Yaskawa INFORM job: BLACKRUN.JBI

/JOB
//NAME BLACKRUN
//POS
///NPOS 4041,0,0,0,0,0
///TOOL 0
///POSTYPE PULSE
///PULSE
C00000=-2822,58859,-1118,-1041,-34109,-89
C00001=-2591,62265,5411,-1016,-36162,-226
C00002=-2591,62265,4011,-1016,-36162,-226
C00003=-2454,62257,4002,-1034,-36158,-281
C00004=-2454,62257,5402,-1034,-36158,-281
C00005=-2634,62224,5347,-1011,-36136,-208
C00006=-2634,62224,3947,-1011,-36136,-208
C00007=-2403,62210,3931,-1041,-36129,-301
C00008=-2403,62210,5331,-1041,-36129,-301
C00009=-2660,62181,5282,-1008,-36110,-197
C00010=-2660,62181,3882,-1008,-36110,-197
C00011=-2607,62178,3878,-1015,-36108,-219
C00012=-2607,62178,5278,-1015,-36108,-219
C00013=-2442,62168,5267,-1037,-36104,-285
C00014=-2442,62168,3867,-1037,-36104,-285
C00015=-2393,62165,3864,-1043,-36102,-305
C00016=-2393,62165,5264,-1043,-36102,-305
C00017=-4693,62262,5357,-741,-36142,620
C00018=-4693,62262,3957,-741,-36142,620
C00019=-4619,62257,3952,-751,-36140,591
C00020=-4619,62257,5352,-751,-36140,591
C00021=-4342,62240,5333,-787,-36132,479
C00022=-4342,62240,3933,-787,-36132,479
C00023=-3994,62219,3908,-833,-36122,340
C00024=-3994,62219,5308,-833,-36122,340
C00025=-2682,62138,5217,-1006,-36083,-188
C00026=-2682,62138,3817,-1006,-36083,-188
C00027=-2632,62135,3813,-1012,-36082,-208
C00028=-2632,62135,5213,-1012,-36082,-208
C00029=-2432,62123,5199,-1039,-36076,-288
C00030=-2432,62123,3799,-1039,-36076,-288
C00031=-2387,62120,3796,-1045,-36075,-307
C00032=-2387,62120,5196,-1045,-36075,-307
C00033=-4830,62226,5300,-724,-36119,676
C00034=-4830,62226,3900,-724,-36119,676
C00035=-4543,62208,3880,-762,-36110,560
C00036=-4543,62208,5280,-762,-36110,560
C00037=-4469,62203,5275,-771,-36108,531
C00038=-4469,62203,3875,-771,-36108,531
C00039=-4244,62190,3859,-801,-36102,441
C00040=-4244,62190,5259,-801,-36102,441
C00041=-4090,62180,5248,-821,-36097,379
C00042=-4090,62180,3848,-821,-36097,379
C00043=-3855,62166,3832,-852,-36090,284
C00044=-3855,62166,5232,-852,-36090,284
C00045=-2696,62095,5151,-1005,-36057,-182
C00046=-2696,62095,3751,-1005,-36057,-182
C00047=-2654,62092,3748,-1010,-36056,-198
C00048=-2654,62092,5148,-1010,-36056,-198
C00049=-2423,62078,5132,-1041,-36049,-292
C00050=-2423,62078,3732,-1041,-36049,-292
C00051=-2381,62075,3729,-1046,-36048,-309
C00052=-2381,62075,5129,-1046,-36048,-309
C00053=-4912,62186,5238,-714,-36094,710
C00054=-4912,62186,3838,-714,-36094,710
C00055=-4782,62178,3829,-731,-36090,657
C00056=-4782,62178,5229,-731,-36090,657
C00057=-4596,62167,5216,-755,-36085,583
C00058=-4596,62167,3816,-755,-36085,583
C00059=-4445,62157,3806,-775,-36081,522
C00060=-4445,62157,5206,-775,-36081,522
C00061=-3929,62126,5170,-843,-36066,315
C00062=-3929,62126,3770,-843,-36066,315
C00063=-3778,62117,3759,-863,-36061,254
C00064=-3778,62117,5159,-863,-36061,254
C00065=-2708,62051,5084,-1004,-36030,-176
C00066=-2708,62051,3684,-1004,-36030,-176
C00067=-2673,62049,3682,-1008,-36029,-191
C00068=-2673,62049,5082,-1008,-36029,-191
C00069=-2413,62033,5064,-1043,-36022,-295
C00070=-2413,62033,3664,-1043,-36022,-295
C00071=-2371,62031,3661,-1048,-36020,-312
C00072=-2371,62031,5061,-1048,-36020,-312
C00073=-4976,62146,5176,-706,-36069,736
C00074=-4976,62146,3776,-706,-36069,736
C00075=-4864,62139,3768,-721,-36066,691
C00076=-4864,62139,5168,-721,-36066,691
C00077=-4713,62129,5157,-740,-36062,630
C00078=-4713,62129,3757,-740,-36062,630
C00079=-4576,62121,3748,-758,-36058,575
C00080=-4576,62121,5148,-758,-36058,575
C00081=-4488,62116,5142,-770,-36055,540
C00082=-4488,62116,3742,-770,-36055,540
C00083=-4415,62111,3737,-780,-36053,510
C00084=-4415,62111,5137,-780,-36053,510
C00085=-3821,62075,5095,-858,-36036,272
C00086=-3821,62075,3695,-858,-36036,272
C00087=-3713,62068,3688,-872,-36032,228
C00088=-3713,62068,5088,-872,-36032,228
C00089=-2726,62008,5019,-1002,-36004,-168
C00090=-2726,62008,3619,-1002,-36004,-168
C00091=-2688,62006,3616,-1007,-36003,-184
C00092=-2688,62006,5016,-1007,-36003,-184
C00093=-2407,61988,4996,-1044,-35994,-297
C00094=-2407,61988,3596,-1044,-35994,-297
C00095=-2361,61986,3593,-1050,-35993,-315
C00096=-2361,61986,4993,-1050,-35993,-315
C00097=-5012,62103,5111,-702,-36043,751
C00098=-5012,62103,3711,-702,-36043,751
C00099=-4928,62098,3705,-713,-36041,717
C00100=-4928,62098,5105,-713,-36041,717
C00101=-3752,62026,5023,-868,-36007,244
C00102=-3752,62026,3623,-868,-36007,244
C00103=-3661,62021,3617,-880,-36004,208
C00104=-3661,62021,5017,-880,-36004,208
C00105=-2738,61964,4952,-1001,-35977,-163
C00106=-2738,61964,3552,-1001,-35977,-163
C00107=-2699,61962,3550,-1006,-35976,-179
C00108=-2699,61962,4950,-1006,-35976,-179
C00109=-2401,61944,4929,-1046,-35967,-299
C00110=-2401,61944,3529,-1046,-35967,-299
C00111=-2355,61941,3526,-1052,-35966,-317
C00112=-2355,61941,4926,-1052,-35966,-317
C00113=-5056,62061,5047,-697,-36018,769
C00114=-5056,62061,3647,-697,-36018,769
C00115=-4985,62057,3642,-706,-36016,741
C00116=-4985,62057,5042,-706,-36016,741
C00117=-3697,61979,4952,-876,-35978,223
C00118=-3697,61979,3552,-876,-35978,223
C00119=-3630,61975,3548,-884,-35976,196
C00120=-3630,61975,4948,-884,-35976,196
C00121=-2745,61921,4886,-1001,-35950,-160
C00122=-2745,61921,3486,-1001,-35950,-160
C00123=-2714,61919,3484,-1005,-35949,-172
C00124=-2714,61919,4884,-1005,-35949,-172
C00125=-2398,61899,4862,-1047,-35940,-299
C00126=-2398,61899,3462,-1047,-35940,-299
C00127=-2352,61897,3458,-1053,-35939,-318
C00128=-2352,61897,4858,-1053,-35939,-318
C00129=-5099,62020,4983,-692,-35992,787
C00130=-5099,62020,3583,-692,-35992,787
C00131=-5025,62015,3578,-701,-35990,757
C00132=-5025,62015,4978,-701,-35990,757
C00133=-3656,61932,4882,-882,-35950,207
C00134=-3656,61932,3482,-882,-35950,207
C00135=-3603,61929,3479,-889,-35948,186
C00136=-3603,61929,4879,-889,-35948,186
C00137=-2750,61877,4819,-1001,-35923,-157
C00138=-2750,61877,3419,-1001,-35923,-157
C00139=-2722,61875,3417,-1005,-35922,-169
C00140=-2722,61875,4817,-1005,-35922,-169
C00141=-2392,61855,4794,-1048,-35913,-301
C00142=-2392,61855,3394,-1048,-35913,-301
C00143=-2343,61852,3391,-1055,-35911,-321
C00144=-2343,61852,4791,-1055,-35911,-321
C00145=126,61702,4618,-1380,-35839,-1313
C00146=126,61702,3218,-1380,-35839,-1313
C00147=150,61700,3217,-1383,-35838,-1323
C00148=150,61700,4617,-1383,-35838,-1323
C00149=-5135,61977,4919,-688,-35966,802
C00150=-5135,61977,3519,-688,-35966,802
C00151=-5065,61973,3514,-697,-35964,773
C00152=-5065,61973,4914,-697,-35964,773
C00153=-3632,61886,4814,-886,-35922,198
C00154=-3632,61886,3414,-886,-35922,198
C00155=-3565,61882,3409,-894,-35920,171
C00156=-3565,61882,4809,-894,-35920,171
C00157=-2758,61833,4753,-1001,-35896,-154
C00158=-2758,61833,3353,-1001,-35896,-154
C00159=-2726,61831,3350,-1005,-35896,-166
C00160=-2726,61831,4750,-1005,-35896,-166
C00161=-2389,61810,4727,-1049,-35886,-302
C00162=-2389,61810,3327,-1049,-35886,-302
C00163=-2350,61808,3324,-1055,-35884,-317
C00164=-2350,61808,4724,-1055,-35884,-317
C00165=-935,61722,4625,-1241,-35843,-886
C00166=-935,61722,3225,-1241,-35843,-886
C00167=-890,61719,3222,-1247,-35842,-904
C00168=-890,61719,4622,-1247,-35842,-904
C00169=128,61657,4551,-1381,-35812,-1313
C00170=128,61657,3151,-1381,-35812,-1313
C00171=171,61655,3148,-1387,-35811,-1330
C00172=171,61655,4548,-1387,-35811,-1330
C00173=-5164,61935,4854,-684,-35940,814
C00174=-5164,61935,3454,-684,-35940,814
C00175=-5104,61931,3449,-692,-35938,790
C00176=-5104,61931,4849,-692,-35938,790
C00177=-3601,61840,4744,-890,-35894,186
C00178=-3601,61840,3344,-890,-35894,186
C00179=-3528,61835,3339,-900,-35892,156
C00180=-3528,61835,4739,-900,-35892,156
C00181=-2766,61789,4686,-1001,-35870,-150
C00182=-2766,61789,3286,-1001,-35870,-150
C00183=-2730,61787,3284,-1005,-35869,-164
C00184=-2730,61787,4684,-1005,-35869,-164
C00185=-936,61678,4558,-1242,-35816,-885
C00186=-936,61678,3158,-1242,-35816,-885
C00187=-891,61675,3155,-1248,-35815,-903
C00188=-891,61675,4555,-1248,-35815,-903
C00189=-747,61666,4545,-1267,-35810,-961
C00190=-747,61666,3145,-1267,-35810,-961
C00191=-704,61664,3142,-1272,-35809,-978
C00192=-704,61664,4542,-1272,-35809,-978
C00193=142,61613,4483,-1384,-35784,-1318
C00194=142,61613,3083,-1384,-35784,-1318
C00195=180,61610,3080,-1389,-35783,-1333
C00196=180,61610,4480,-1389,-35783,-1333
C00197=-5196,61892,4789,-681,-35914,827
C00198=-5196,61892,3389,-681,-35914,827
C00199=-5140,61889,3385,-688,-35912,805
C00200=-5140,61889,4785,-688,-35912,805
C00201=-3560,61793,4675,-896,-35866,170
C00202=-3560,61793,3275,-896,-35866,170
C00203=-3500,61789,3270,-904,-35864,146
C00204=-3500,61789,4670,-904,-35864,146
C00205=-2766,61745,4619,-1001,-35843,-149
C00206=-2766,61745,3219,-1001,-35843,-149
C00207=-2735,61743,3217,-1005,-35842,-162
C00208=-2735,61743,4617,-1005,-35842,-162
C00209=-2205,61711,4580,-1075,-35826,-375
C00210=-2205,61711,3180,-1075,-35826,-375
C00211=-2117,61705,3174,-1087,-35824,-410
C00212=-2117,61705,4574,-1087,-35824,-410
C00213=-937,61634,4491,-1242,-35789,-884
C00214=-937,61634,3091,-1242,-35789,-884
C00215=-891,61631,3088,-1248,-35787,-902
C00216=-891,61631,4488,-1248,-35787,-902
C00217=-737,61622,4477,-1269,-35783,-964
C00218=-737,61622,3077,-1269,-35783,-964
C00219=-688,61619,3074,-1275,-35782,-984
C00220=-688,61619,4474,-1275,-35782,-984
C00221=-333,61597,4449,-1322,-35771,-1127
C00222=-333,61597,3049,-1322,-35771,-1127
C00223=-294,61595,3047,-1327,-35770,-1142
C00224=-294,61595,4447,-1327,-35770,-1142
C00225=155,61568,4415,-1386,-35757,-1323
C00226=155,61568,3015,-1386,-35757,-1323
C00227=197,61565,3012,-1392,-35755,-1340
C00228=197,61565,4412,-1392,-35755,-1340
C00229=-5222,61849,4723,-678,-35888,838
C00230=-5222,61849,3323,-678,-35888,838
C00231=-5162,61845,3319,-686,-35886,814
C00232=-5162,61845,4719,-686,-35886,814
C00233=-3529,61747,4605,-901,-35838,158
C00234=-3529,61747,3205,-901,-35838,158
C00235=-3470,61743,3201,-909,-35836,134
C00236=-3470,61743,4601,-909,-35836,134
C00237=-2767,61701,4552,-1002,-35816,-148
C00238=-2767,61701,3152,-1002,-35816,-148
C00239=-2732,61698,3150,-1006,-35815,-162
C00240=-2732,61698,4550,-1006,-35815,-162
C00241=-2237,61668,4515,-1072,-35800,-361
C00242=-2237,61668,3115,-1072,-35800,-361
C00243=-2163,61664,3110,-1081,-35798,-391
C00244=-2163,61664,4510,-1081,-35798,-391
C00245=-2146,61663,4509,-1084,-35797,-398
C00246=-2146,61663,3109,-1084,-35797,-398
C00247=-2090,61659,3105,-1091,-35796,-420
C00248=-2090,61659,4505,-1091,-35796,-420
C00249=-1893,61648,4491,-1117,-35790,-499
C00250=-1893,61648,3091,-1117,-35790,-499
C00251=-1858,61645,3089,-1122,-35789,-513
C00252=-1858,61645,4489,-1122,-35789,-513
C00253=-1731,61638,4480,-1138,-35785,-564
C00254=-1731,61638,3080,-1138,-35785,-564
C00255=-1605,61630,3071,-1155,-35781,-615
C00256=-1605,61630,4471,-1155,-35781,-615
C00257=-934,61590,4424,-1243,-35762,-884
C00258=-934,61590,3024,-1243,-35762,-884
C00259=-892,61587,3021,-1249,-35760,-901
C00260=-892,61587,4421,-1249,-35760,-901
C00261=-730,61577,4410,-1270,-35756,-966
C00262=-730,61577,3010,-1270,-35756,-966
C00263=-674,61574,3006,-1278,-35754,-989
C00264=-674,61574,4406,-1278,-35754,-989
C00265=-425,61559,4389,-1311,-35747,-1089
C00266=-425,61559,2989,-1311,-35747,-1089
C00267=-351,61554,2984,-1320,-35744,-1119
C00268=-351,61554,4384,-1320,-35744,-1119
C00269=-309,61552,4381,-1326,-35743,-1136
C00270=-309,61552,2981,-1326,-35743,-1136
C00271=-270,61549,2978,-1331,-35742,-1151
C00272=-270,61549,4378,-1331,-35742,-1151
C00273=-151,61542,4370,-1347,-35739,-1199
C00274=-151,61542,2970,-1347,-35739,-1199
C00275=-102,61539,2966,-1353,-35737,-1219
C00276=-102,61539,4366,-1353,-35737,-1219
C00277=169,61523,4347,-1389,-35729,-1327
C00278=169,61523,2947,-1389,-35729,-1327
C00279=204,61521,2945,-1394,-35728,-1342
C00280=204,61521,4345,-1394,-35728,-1342
C00281=-5244,61806,4658,-676,-35862,848
C00282=-5244,61806,3258,-676,-35862,848
C00283=-5188,61802,3254,-683,-35860,825
C00284=-5188,61802,4654,-683,-35860,825
C00285=-3502,61701,4536,-906,-35810,148
C00286=-3502,61701,3136,-906,-35810,148
C00287=-3442,61697,3132,-913,-35808,124
C00288=-3442,61697,4532,-913,-35808,124
C00289=-2765,61656,4485,-1003,-35788,-148
C00290=-2765,61656,3085,-1003,-35788,-148
C00291=-2733,61654,3083,-1007,-35788,-161
C00292=-2733,61654,4483,-1007,-35788,-161
C00293=-2262,61626,4450,-1069,-35774,-350
C00294=-2262,61626,3050,-1069,-35774,-350
C00295=-2217,61623,3047,-1075,-35772,-369
C00296=-2217,61623,4447,-1075,-35772,-369
C00297=-2108,61616,4439,-1089,-35769,-412
C00298=-2108,61616,3039,-1089,-35769,-412
C00299=-2034,61612,3034,-1099,-35767,-442
C00300=-2034,61612,4434,-1099,-35767,-442
C00301=-1890,61603,4424,-1118,-35763,-500
C00302=-1890,61603,3024,-1118,-35763,-500
C00303=-1848,61601,3021,-1124,-35761,-517
C00304=-1848,61601,4421,-1124,-35761,-517
C00305=-1760,61595,4415,-1135,-35759,-552
C00306=-1760,61595,3015,-1135,-35759,-552
C00307=-1693,61591,3010,-1144,-35757,-579
C00308=-1693,61591,4410,-1144,-35757,-579
C00309=-1634,61588,4406,-1152,-35755,-603
C00310=-1634,61588,3006,-1152,-35755,-603
C00311=-1574,61584,3002,-1160,-35753,-627
C00312=-1574,61584,4402,-1160,-35753,-627
C00313=-928,61545,4357,-1245,-35734,-886
C00314=-928,61545,2957,-1245,-35734,-886
C00315=-889,61543,2954,-1250,-35733,-902
C00316=-889,61543,4354,-1250,-35733,-902
C00317=-728,61533,4343,-1271,-35728,-967
C00318=-728,61533,2943,-1271,-35728,-967
C00319=-643,61528,2937,-1283,-35726,-1001
C00320=-643,61528,4337,-1283,-35726,-1001
C00321=-454,61516,4324,-1308,-35720,-1077
C00322=-454,61516,2924,-1308,-35720,-1077
C00323=-390,61513,2919,-1316,-35719,-1102
C00324=-390,61513,4319,-1316,-35719,-1102
C00325=-359,61511,4317,-1320,-35718,-1115
C00326=-359,61511,2917,-1320,-35718,-1115
C00327=-338,61509,2916,-1323,-35717,-1123
C00328=-338,61509,4316,-1323,-35717,-1123
C00329=-285,61506,4312,-1330,-35715,-1145
C00330=-285,61506,2912,-1330,-35715,-1145
C00331=-250,61504,2910,-1334,-35714,-1159
C00332=-250,61504,4310,-1334,-35714,-1159
C00333=-145,61498,4302,-1348,-35711,-1201
C00334=-145,61498,2902,-1348,-35711,-1201
C00335=-103,61495,2899,-1354,-35710,-1218
C00336=-103,61495,4299,-1354,-35710,-1218
C00337=175,61478,4280,-1390,-35702,-1329
C00338=175,61478,2880,-1390,-35702,-1329
C00339=214,61476,2877,-1396,-35701,-1345
C00340=214,61476,4277,-1396,-35701,-1345
C00341=-5263,61762,4592,-674,-35835,856
C00342=-5263,61762,3192,-674,-35835,856
C00343=-5217,61760,3189,-680,-35834,837
C00344=-5217,61760,4589,-680,-35834,837
C00345=-3471,61654,4467,-910,-35782,136
C00346=-3471,61654,3067,-910,-35782,136
C00347=-3412,61651,3063,-918,-35781,112
C00348=-3412,61651,4463,-918,-35781,112
C00349=-2765,61612,4418,-1003,-35761,-148
C00350=-2765,61612,3018,-1003,-35761,-148
C00351=-2734,61610,3016,-1008,-35761,-160
C00352=-2734,61610,4416,-1008,-35761,-160
C00353=-2281,61583,4384,-1067,-35747,-342
C00354=-2281,61583,2984,-1067,-35747,-342
C00355=-2235,61580,2981,-1073,-35746,-361
C00356=-2235,61580,4381,-1073,-35746,-361
C00357=-2077,61570,4370,-1094,-35741,-424
C00358=-2077,61570,2970,-1094,-35741,-424
C00359=-2024,61567,2966,-1101,-35740,-445
C00360=-2024,61567,4366,-1101,-35740,-445
C00361=-1884,61559,4356,-1120,-35735,-502
C00362=-1884,61559,2956,-1120,-35735,-502
C00363=-1838,61556,2953,-1126,-35734,-520
C00364=-1838,61556,4353,-1126,-35734,-520
C00365=-1782,61552,4349,-1133,-35732,-543
C00366=-1782,61552,2949,-1133,-35732,-543
C00367=-1740,61550,2946,-1139,-35731,-560
C00368=-1740,61550,4346,-1139,-35731,-560
C00369=-1603,61542,4337,-1157,-35727,-615
C00370=-1603,61542,2937,-1157,-35727,-615
C00371=-1554,61539,2933,-1163,-35726,-634
C00372=-1554,61539,4333,-1163,-35726,-634
C00373=-925,61501,4290,-1246,-35707,-887
C00374=-925,61501,2890,-1246,-35707,-887
C00375=-886,61498,2887,-1251,-35706,-902
C00376=-886,61498,4287,-1251,-35706,-902
C00377=-725,61489,4276,-1273,-35701,-967
C00378=-725,61489,2876,-1273,-35701,-967
C00379=-693,61487,2873,-1277,-35700,-980
C00380=-693,61487,4273,-1277,-35700,-980
C00381=-676,61486,4272,-1279,-35700,-987
C00382=-676,61486,2872,-1279,-35700,-987
C00383=-623,61483,2869,-1286,-35698,-1008
C00384=-623,61483,4269,-1286,-35698,-1008
C00385=-472,61473,4258,-1306,-35694,-1069
C00386=-472,61473,2858,-1306,-35694,-1069
C00387=-423,61470,2855,-1312,-35692,-1089
C00388=-423,61470,4255,-1312,-35692,-1089
C00389=-268,61461,4244,-1333,-35688,-1151
C00390=-268,61461,2844,-1333,-35688,-1151
C00391=-226,61459,2841,-1338,-35687,-1168
C00392=-226,61459,4241,-1338,-35687,-1168
C00393=-138,61453,4235,-1350,-35684,-1203
C00394=-138,61453,2835,-1350,-35684,-1203
C00395=-100,61451,2832,-1355,-35683,-1218
C00396=-100,61451,4232,-1355,-35683,-1218
C00397=181,61434,4212,-1392,-35674,-1331
C00398=181,61434,2812,-1392,-35674,-1331
C00399=220,61432,2810,-1397,-35673,-1347
C00400=220,61432,4210,-1397,-35673,-1347
C00401=-5288,61720,4527,-671,-35809,866
C00402=-5288,61720,3127,-671,-35809,866
C00403=-5236,61716,3123,-678,-35807,845
C00404=-5236,61716,4523,-678,-35807,845
C00405=-3448,61609,4398,-914,-35755,127
C00406=-3448,61609,2998,-914,-35755,127
C00407=-3385,61605,2994,-922,-35753,102
C00408=-3385,61605,4394,-922,-35753,102
C00409=-2763,61567,4351,-1004,-35734,-148
C00410=-2763,61567,2951,-1004,-35734,-148
C00411=-2731,61565,2948,-1009,-35733,-161
C00412=-2731,61565,4348,-1009,-35733,-161
C00413=-2296,61539,4318,-1066,-35721,-336
C00414=-2296,61539,2918,-1066,-35721,-336
C00415=-2254,61537,2915,-1072,-35719,-353
C00416=-2254,61537,4315,-1072,-35719,-353
C00417=-2067,61525,4302,-1096,-35714,-427
C00418=-2067,61525,2902,-1096,-35714,-427
C00419=-2015,61522,2899,-1103,-35712,-449
C00420=-2015,61522,4299,-1103,-35712,-449
C00421=-1871,61514,4288,-1122,-35708,-506
C00422=-1871,61514,2888,-1122,-35708,-506
C00423=-1829,61511,2886,-1128,-35707,-523
C00424=-1829,61511,4286,-1128,-35707,-523
C00425=-1797,61509,4283,-1132,-35706,-536
C00426=-1797,61509,2883,-1132,-35706,-536
C00427=-1758,61507,2881,-1137,-35705,-552
C00428=-1758,61507,4281,-1137,-35705,-552
C00429=-1579,61496,4268,-1161,-35699,-624
C00430=-1579,61496,2868,-1161,-35699,-624
C00431=-1533,61493,2865,-1167,-35698,-642
C00432=-1533,61493,4265,-1167,-35698,-642
C00433=-922,61456,4222,-1247,-35680,-887
C00434=-922,61456,2822,-1247,-35680,-887
C00435=-880,61454,2819,-1253,-35679,-904
C00436=-880,61454,4219,-1253,-35679,-904
C00437=-719,61444,4208,-1274,-35674,-969
C00438=-719,61444,2808,-1274,-35674,-969
C00439=-687,61442,2806,-1278,-35673,-982
C00440=-687,61442,4206,-1278,-35673,-982
C00441=-652,61440,4204,-1283,-35672,-996
C00442=-652,61440,2804,-1283,-35672,-996
C00443=-603,61437,2800,-1289,-35670,-1016
C00444=-603,61437,4200,-1289,-35670,-1016
C00445=-483,61430,4192,-1305,-35667,-1064
C00446=-483,61430,2792,-1305,-35667,-1064
C00447=-441,61427,2789,-1311,-35666,-1081
C00448=-441,61427,4189,-1311,-35666,-1081
C00449=-251,61416,4176,-1336,-35660,-1157
C00450=-251,61416,2776,-1336,-35660,-1157
C00451=-213,61414,2773,-1341,-35659,-1172
C00452=-213,61414,4173,-1341,-35659,-1172
C00453=-135,61409,4168,-1351,-35657,-1203
C00454=-135,61409,2768,-1351,-35657,-1203
C00455=-97,61407,2765,-1356,-35656,-1219
C00456=-97,61407,4165,-1356,-35656,-1219
C00457=188,61390,4145,-1394,-35647,-1333
C00458=188,61390,2745,-1394,-35647,-1333
C00459=226,61387,2742,-1399,-35646,-1349
C00460=226,61387,4142,-1399,-35646,-1349
C00461=-5310,61676,4461,-669,-35783,876
C00462=-5310,61676,3061,-669,-35783,876
C00463=-5261,61673,3058,-675,-35781,856
C00464=-5261,61673,4458,-675,-35781,856
C00465=-3421,61563,4329,-918,-35727,117
C00466=-3421,61563,2929,-918,-35727,117
C00467=-3354,61559,2925,-927,-35725,90
C00468=-3354,61559,4325,-927,-35725,90
C00469=-2760,61523,4283,-1006,-35707,-149
C00470=-2760,61523,2883,-1006,-35707,-149
C00471=-2725,61521,2881,-1010,-35706,-163
C00472=-2725,61521,4281,-1010,-35706,-163
C00473=-2304,61495,4252,-1066,-35694,-332
C00474=-2304,61495,2852,-1066,-35694,-332
C00475=-2265,61493,2849,-1071,-35693,-348
C00476=-2265,61493,4249,-1071,-35693,-348
C00477=-2065,61481,4235,-1097,-35687,-428
C00478=-2065,61481,2835,-1097,-35687,-428
C00479=-2008,61478,2831,-1105,-35685,-451
C00480=-2008,61478,4231,-1105,-35685,-451
C00481=-1861,61469,4221,-1124,-35681,-510
C00482=-1861,61469,2821,-1124,-35681,-510
C00483=-1770,61463,2814,-1136,-35678,-546
C00484=-1770,61463,4214,-1136,-35678,-546
C00485=-1562,61451,4200,-1164,-35672,-630
C00486=-1562,61451,2800,-1164,-35672,-630
C00487=-1520,61448,2797,-1169,-35671,-647
C00488=-1520,61448,4197,-1169,-35671,-647
C00489=-916,61412,4155,-1249,-35653,-889
C00490=-916,61412,2755,-1249,-35653,-889
C00491=-870,61409,2752,-1255,-35651,-908
C00492=-870,61409,4152,-1255,-35651,-908
C00493=-716,61400,4141,-1275,-35647,-970
C00494=-716,61400,2741,-1275,-35647,-970
C00495=-684,61398,2739,-1279,-35646,-982
C00496=-684,61398,4139,-1279,-35646,-982
C00497=-631,61395,4135,-1286,-35644,-1004
C00498=-631,61395,2735,-1286,-35644,-1004
C00499=-575,61391,2731,-1294,-35643,-1026
C00500=-575,61391,4131,-1294,-35643,-1026
C00501=-487,61386,4125,-1305,-35640,-1061
C00502=-487,61386,2725,-1305,-35640,-1061
C00503=-449,61384,2722,-1311,-35639,-1077
C00504=-449,61384,4122,-1311,-35639,-1077
C00505=-238,61371,4108,-1338,-35633,-1162
C00506=-238,61371,2708,-1338,-35633,-1162
C00507=-203,61369,2705,-1343,-35632,-1176
C00508=-203,61369,4105,-1343,-35632,-1176
C00509=-129,61365,4100,-1353,-35629,-1205
C00510=-129,61365,2700,-1353,-35629,-1205
C00511=-87,61362,2697,-1358,-35628,-1222
C00512=-87,61362,4097,-1358,-35628,-1222
C00513=198,61345,4077,-1396,-35620,-1337
C00514=198,61345,2677,-1396,-35620,-1337
C00515=233,61343,2675,-1400,-35619,-1351
C00516=233,61343,4075,-1400,-35619,-1351
C00517=-5329,61633,4395,-667,-35756,884
C00518=-5329,61633,2995,-667,-35756,884
C00519=-5283,61630,2992,-673,-35755,865
C00520=-5283,61630,4392,-673,-35755,865
C00521=-3390,61516,4260,-923,-35699,105
C00522=-3390,61516,2860,-923,-35699,105
C00523=-3330,61513,2856,-931,-35697,81
C00524=-3330,61513,4256,-931,-35697,81
C00525=-2754,61478,4216,-1007,-35680,-150
C00526=-2754,61478,2816,-1007,-35680,-150
C00527=-2722,61476,2814,-1011,-35679,-163
C00528=-2722,61476,4214,-1011,-35679,-163
C00529=-2311,61452,4185,-1065,-35667,-328
C00530=-2311,61452,2785,-1065,-35667,-328
C00531=-2273,61449,2782,-1071,-35666,-344
C00532=-2273,61449,4182,-1071,-35666,-344
C00533=-2072,61437,4168,-1097,-35660,-424
C00534=-2072,61437,2768,-1097,-35660,-424
C00535=-2002,61433,2764,-1106,-35658,-452
C00536=-2002,61433,4164,-1106,-35658,-452
C00537=-1851,61424,4153,-1126,-35653,-513
C00538=-1851,61424,2753,-1126,-35653,-513
C00539=-1781,61420,2748,-1135,-35651,-541
C00540=-1781,61420,4148,-1135,-35651,-541
C00541=-1549,61406,4132,-1166,-35644,-634
C00542=-1549,61406,2732,-1166,-35644,-634
C00543=-1510,61404,2729,-1171,-35643,-650
C00544=-1510,61404,4129,-1171,-35643,-650
C00545=-906,61367,4087,-1251,-35625,-893
C00546=-906,61367,2687,-1251,-35625,-893
C00547=-861,61365,2684,-1257,-35624,-911
C00548=-861,61365,4084,-1257,-35624,-911
C00549=-713,61356,4074,-1276,-35620,-970
C00550=-713,61356,2674,-1276,-35620,-970
C00551=-681,61354,2672,-1281,-35619,-983
C00552=-681,61354,4072,-1281,-35619,-983
C00553=-608,61349,4066,-1290,-35616,-1013
C00554=-608,61349,2666,-1290,-35616,-1013
C00555=-558,61346,2663,-1297,-35615,-1032
C00556=-558,61346,4063,-1297,-35615,-1032
C00557=-495,61343,4059,-1305,-35613,-1058
C00558=-495,61343,2659,-1305,-35613,-1058
C00559=-453,61340,2656,-1311,-35612,-1075
C00560=-453,61340,4056,-1311,-35612,-1075
C00561=-225,61326,4040,-1341,-35605,-1166
C00562=-225,61326,2640,-1341,-35605,-1166
C00563=-193,61324,2637,-1345,-35604,-1179
C00564=-193,61324,4037,-1345,-35604,-1179
C00565=-123,61320,4033,-1354,-35602,-1207
C00566=-123,61320,2633,-1354,-35602,-1207
C00567=-84,61318,2630,-1359,-35601,-1223
C00568=-84,61318,4030,-1359,-35601,-1223
C00569=204,61301,4010,-1397,-35592,-1339
C00570=204,61301,2610,-1397,-35592,-1339
C00571=239,61298,2607,-1402,-35591,-1353
C00572=239,61298,4007,-1402,-35591,-1353
C00573=-5351,61590,4330,-665,-35730,893
C00574=-5351,61590,2930,-665,-35730,893
C00575=-5302,61587,2926,-671,-35729,873
C00576=-5302,61587,4326,-671,-35729,873
C00577=-3363,61471,4191,-927,-35671,95
C00578=-3363,61471,2791,-927,-35671,95
C00579=-3320,61468,2788,-933,-35670,78
C00580=-3320,61468,4188,-933,-35670,78
C00581=-2751,61434,4149,-1008,-35653,-151
C00582=-2751,61434,2749,-1008,-35653,-151
C00583=-2720,61432,2747,-1012,-35652,-164
C00584=-2720,61432,4147,-1012,-35652,-164
C00585=-2319,61408,4119,-1065,-35640,-325
C00586=-2319,61408,2719,-1065,-35640,-325
C00587=-2281,61406,2716,-1070,-35639,-340
C00588=-2281,61406,4116,-1070,-35639,-340
C00589=-2070,61393,4101,-1098,-35633,-425
C00590=-2070,61393,2701,-1098,-35633,-425
C00591=-1996,61389,2696,-1108,-35630,-454
C00592=-1996,61389,4096,-1108,-35630,-454
C00593=-1845,61379,4086,-1128,-35626,-515
C00594=-1845,61379,2686,-1128,-35626,-515
C00595=-1789,61376,2682,-1135,-35624,-538
C00596=-1789,61376,4082,-1135,-35624,-538
C00597=-1539,61361,4064,-1168,-35617,-638
C00598=-1539,61361,2664,-1168,-35617,-638
C00599=-1501,61359,2662,-1173,-35616,-653
C00600=-1501,61359,4062,-1173,-35616,-653
C00601=-893,61322,4019,-1253,-35598,-897
C00602=-893,61322,2619,-1253,-35598,-897
C00603=-851,61320,2616,-1259,-35596,-914
C00604=-851,61320,4016,-1259,-35596,-914
C00605=-717,61312,4007,-1277,-35593,-968
C00606=-717,61312,2607,-1277,-35593,-968
C00607=-689,61310,2605,-1280,-35592,-979
C00608=-689,61310,4005,-1280,-35592,-979
C00609=-591,61304,3998,-1293,-35589,-1019
C00610=-591,61304,2598,-1293,-35589,-1019
C00611=-542,61301,2595,-1300,-35587,-1038
C00612=-542,61301,3995,-1300,-35587,-1038
C00613=-496,61299,3992,-1306,-35586,-1057
C00614=-496,61299,2592,-1306,-35586,-1057
C00615=-450,61296,2588,-1312,-35585,-1075
C00616=-450,61296,3988,-1312,-35585,-1075
C00617=-218,61282,3972,-1342,-35578,-1168
C00618=-218,61282,2572,-1342,-35578,-1168
C00619=-187,61280,2570,-1347,-35577,-1181
C00620=-187,61280,3970,-1347,-35577,-1181
C00621=-116,61276,3965,-1356,-35575,-1209
C00622=-116,61276,2565,-1356,-35575,-1209
C00623=-78,61273,2562,-1361,-35574,-1225
C00624=-78,61273,3962,-1361,-35574,-1225
C00625=207,61256,3943,-1399,-35565,-1339
C00626=207,61256,2543,-1399,-35565,-1339
C00627=242,61254,2540,-1403,-35564,-1353
C00628=242,61254,3940,-1403,-35564,-1353
C00629=-5370,61546,4264,-663,-35704,901
C00630=-5370,61546,2864,-663,-35704,901
C00631=-5320,61543,2861,-670,-35702,881
C00632=-5320,61543,4261,-670,-35702,881
C00633=-3349,61425,4123,-930,-35644,90
C00634=-3349,61425,2723,-930,-35644,90
C00635=-3300,61422,2720,-936,-35642,70
C00636=-3300,61422,4120,-936,-35642,70
C00637=-2749,61389,4082,-1009,-35626,-151
C00638=-2749,61389,2682,-1009,-35626,-151
C00639=-2714,61387,2679,-1014,-35625,-166
C00640=-2714,61387,4079,-1014,-35625,-166
C00641=-2450,61371,4061,-1049,-35617,-271
C00642=-2450,61371,2661,-1049,-35617,-271
C00643=-2425,61370,2659,-1052,-35616,-281
C00644=-2425,61370,4059,-1052,-35616,-281
C00645=-2320,61364,4052,-1066,-35613,-324
C00646=-2320,61364,2652,-1066,-35613,-324
C00647=-2281,61361,2649,-1071,-35612,-339
C00648=-2281,61361,4049,-1071,-35612,-339
C00649=-2074,61349,4035,-1098,-35606,-422
C00650=-2074,61349,2635,-1098,-35606,-422
C00651=-1986,61344,2628,-1110,-35603,-458
C00652=-1986,61344,4028,-1110,-35603,-458
C00653=-1842,61335,4018,-1129,-35599,-516
C00654=-1842,61335,2618,-1129,-35599,-516
C00655=-1786,61332,2614,-1136,-35597,-538
C00656=-1786,61332,4014,-1136,-35597,-538
C00657=-1530,61316,3997,-1170,-35590,-641
C00658=-1530,61316,2597,-1170,-35590,-641
C00659=-1494,61314,2594,-1175,-35589,-655
C00660=-1494,61314,3994,-1175,-35589,-655
C00661=-883,61278,3952,-1255,-35570,-901
C00662=-883,61278,2552,-1255,-35570,-901
C00663=-841,61275,2549,-1261,-35569,-918
C00664=-841,61275,3949,-1261,-35569,-918
C00665=-725,61268,3941,-1276,-35566,-964
C00666=-725,61268,2541,-1276,-35566,-964
C00667=-693,61266,2538,-1281,-35565,-977
C00668=-693,61266,3938,-1281,-35565,-977
C00669=-570,61259,3930,-1297,-35561,-1026
C00670=-570,61259,2530,-1297,-35561,-1026
C00671=-525,61256,2527,-1303,-35560,-1045
C00672=-525,61256,3927,-1303,-35560,-1045
C00673=-490,61254,3924,-1307,-35559,-1059
C00674=-490,61254,2524,-1307,-35559,-1059
C00675=-447,61252,2521,-1313,-35557,-1076
C00676=-447,61252,3921,-1313,-35557,-1076
C00677=-216,61238,3905,-1344,-35550,-1169
C00678=-216,61238,2505,-1344,-35550,-1169
C00679=-177,61235,2502,-1349,-35549,-1184
C00680=-177,61235,3902,-1349,-35549,-1184
C00681=-110,61231,3898,-1357,-35547,-1211
C00682=-110,61231,2498,-1357,-35547,-1211
C00683=-68,61229,2495,-1363,-35546,-1228
C00684=-68,61229,3895,-1363,-35546,-1228
C00685=203,61213,3876,-1399,-35538,-1337
C00686=203,61213,2476,-1399,-35538,-1337
C00687=241,61210,2473,-1404,-35537,-1352
C00688=241,61210,3873,-1404,-35537,-1352
C00689=-5385,61503,4198,-662,-35677,908
C00690=-5385,61503,2798,-662,-35677,908
C00691=-5335,61500,2795,-668,-35676,888
C00692=-5335,61500,4195,-668,-35676,888
C00693=-3336,61380,4055,-932,-35616,85
C00694=-3336,61380,2655,-932,-35616,85
C00695=-3287,61377,2652,-939,-35615,65
C00696=-3287,61377,4052,-939,-35615,65
C00697=-2742,61345,4014,-1011,-35599,-153
C00698=-2742,61345,2614,-1011,-35599,-153
C00699=-2704,61342,2611,-1016,-35597,-169
C00700=-2704,61342,4011,-1016,-35597,-169
C00701=-2454,61328,3994,-1049,-35590,-269
C00702=-2454,61328,2594,-1049,-35590,-269
C00703=-2416,61325,2591,-1054,-35589,-285
C00704=-2416,61325,3991,-1054,-35589,-285
C00705=-2314,61319,3984,-1067,-35586,-326
C00706=-2314,61319,2584,-1067,-35586,-326
C00707=-2279,61317,2582,-1072,-35585,-340
C00708=-2279,61317,3982,-1072,-35585,-340
C00709=-2078,61305,3968,-1098,-35579,-420
C00710=-2078,61305,2568,-1098,-35579,-420
C00711=-2040,61303,2565,-1103,-35578,-436
C00712=-2040,61303,3965,-1103,-35578,-436
C00713=-2019,61301,3964,-1106,-35577,-444
C00714=-2019,61301,2564,-1106,-35577,-444
C00715=-1973,61299,2560,-1112,-35576,-462
C00716=-1973,61299,3960,-1112,-35576,-462
C00717=-1836,61291,3951,-1130,-35572,-517
C00718=-1836,61291,2551,-1130,-35572,-517
C00719=-1787,61288,2547,-1137,-35570,-537
C00720=-1787,61288,3947,-1137,-35570,-537
C00721=-1523,61272,3929,-1172,-35562,-643
C00722=-1523,61272,2529,-1172,-35562,-643
C00723=-1481,61269,2526,-1177,-35561,-660
C00724=-1481,61269,3926,-1177,-35561,-660
C00725=-866,61233,3883,-1258,-35543,-907
C00726=-866,61233,2483,-1258,-35543,-907
C00727=-821,61230,2480,-1264,-35541,-925
C00728=-821,61230,3880,-1264,-35541,-925
C00729=-740,61225,3875,-1275,-35539,-958
C00730=-740,61225,2475,-1275,-35539,-958
C00731=-705,61223,2472,-1280,-35538,-972
C00732=-705,61223,3872,-1280,-35538,-972
C00733=-554,61214,3862,-1300,-35533,-1032
C00734=-554,61214,2462,-1300,-35533,-1032
C00735=-508,61211,2458,-1306,-35532,-1051
C00736=-508,61211,3858,-1306,-35532,-1051
C00737=-480,61209,3856,-1309,-35531,-1062
C00738=-480,61209,2456,-1309,-35531,-1062
C00739=-438,61207,2453,-1315,-35530,-1079
C00740=-438,61207,3853,-1315,-35530,-1079
C00741=-209,61193,3838,-1345,-35523,-1171
C00742=-209,61193,2438,-1345,-35523,-1171
C00743=-178,61191,2435,-1349,-35522,-1183
C00744=-178,61191,3835,-1349,-35522,-1183
C00745=-100,61187,3830,-1360,-35520,-1214
C00746=-100,61187,2430,-1360,-35520,-1214
C00747=-55,61184,2427,-1366,-35519,-1233
C00748=-55,61184,3827,-1366,-35519,-1233
C00749=202,61169,3809,-1399,-35511,-1336
C00750=202,61169,2409,-1399,-35511,-1336
C00751=237,61167,2407,-1404,-35510,-1350
C00752=237,61167,3807,-1404,-35510,-1350
C00753=-5400,61459,4132,-660,-35651,914
C00754=-5400,61459,2732,-660,-35651,914
C00755=-5351,61456,2729,-667,-35649,894
C00756=-5351,61456,4129,-667,-35649,894
C00757=-4929,61431,4099,-723,-35637,725
C00758=-4929,61431,2699,-723,-35637,725
C00759=-4894,61429,2697,-727,-35636,711
C00760=-4894,61429,4097,-727,-35636,711
C00761=-3949,61372,4031,-852,-35608,331
C00762=-3949,61372,2631,-852,-35608,331
C00763=-3878,61368,2626,-861,-35605,303
C00764=-3878,61368,4026,-861,-35605,303
C00765=-3320,61335,3987,-935,-35589,79
C00766=-3320,61335,2587,-935,-35589,79
C00767=-3274,61332,2584,-941,-35587,61
C00768=-3274,61332,3984,-941,-35587,61
C00769=-2733,61300,3946,-1013,-35571,-157
C00770=-2733,61300,2546,-1013,-35571,-157
C00771=-2698,61298,2544,-1017,-35570,-171
C00772=-2698,61298,3944,-1017,-35570,-171
C00773=-2459,61284,3927,-1049,-35563,-267
C00774=-2459,61284,2527,-1049,-35563,-267
C00775=-2417,61281,2524,-1054,-35562,-284
C00776=-2417,61281,3924,-1054,-35562,-284
C00777=-2308,61274,3917,-1069,-35559,-327
C00778=-2308,61274,2517,-1069,-35559,-327
C00779=-2269,61272,2514,-1074,-35557,-343
C00780=-2269,61272,3914,-1074,-35557,-343
C00781=-2083,61261,3901,-1099,-35552,-418
C00782=-2083,61261,2501,-1099,-35552,-418
C00783=-2048,61259,2499,-1103,-35551,-432
C00784=-2048,61259,3899,-1103,-35551,-432
C00785=-2005,61256,3896,-1109,-35550,-449
C00786=-2005,61256,2496,-1109,-35550,-449
C00787=-1963,61254,2493,-1114,-35548,-466
C00788=-1963,61254,3893,-1114,-35548,-466
C00789=-1830,61246,3883,-1132,-35544,-519
C00790=-1830,61246,2483,-1132,-35544,-519
C00791=-1784,61243,2480,-1138,-35543,-538
C00792=-1784,61243,3880,-1138,-35543,-538
C00793=-1517,61227,3862,-1173,-35535,-645
C00794=-1517,61227,2462,-1173,-35535,-645
C00795=-1471,61225,2458,-1179,-35534,-663
C00796=-1471,61225,3858,-1179,-35534,-663
C00797=-846,61187,3815,-1262,-35515,-914
C00798=-846,61187,2415,-1262,-35515,-914
C00799=-726,61180,2407,-1278,-35511,-962
C00800=-726,61180,3807,-1278,-35511,-962
C00801=-540,61169,3794,-1302,-35506,-1037
C00802=-540,61169,2394,-1302,-35506,-1037
C00803=-495,61166,2390,-1308,-35505,-1056
C00804=-495,61166,3790,-1308,-35505,-1056
C00805=-473,61165,3789,-1311,-35504,-1064
C00806=-473,61165,2389,-1311,-35504,-1064
C00807=-421,61162,2385,-1318,-35502,-1085
C00808=-421,61162,3785,-1318,-35502,-1085
C00809=-213,61149,3771,-1345,-35496,-1168
C00810=-213,61149,2371,-1345,-35496,-1168
C00811=-175,61147,2368,-1350,-35495,-1184
C00812=-175,61147,3768,-1350,-35495,-1184
C00813=-87,61142,3762,-1362,-35492,-1219
C00814=-87,61142,2362,-1362,-35492,-1219
C00815=-38,61139,2359,-1369,-35491,-1239
C00816=-38,61139,3759,-1369,-35491,-1239
C00817=198,61125,3742,-1400,-35484,-1334
C00818=198,61125,2342,-1400,-35484,-1334
C00819=236,61123,2340,-1405,-35483,-1349
C00820=236,61123,3740,-1405,-35483,-1349
C00821=-5411,61415,4066,-660,-35624,919
C00822=-5411,61415,2666,-660,-35624,919
C00823=-5366,61413,2663,-666,-35623,901
C00824=-5366,61413,4063,-666,-35623,901
C00825=-4947,61388,4033,-721,-35610,733
C00826=-4947,61388,2633,-721,-35610,733
C00827=-4870,61383,2628,-731,-35608,702
C00828=-4870,61383,4028,-731,-35608,702
C00829=-3967,61329,3965,-850,-35581,339
C00830=-3967,61329,2565,-850,-35581,339
C00831=-3865,61323,2558,-864,-35578,299
C00832=-3865,61323,3958,-864,-35578,299
C00833=-3303,61290,3919,-938,-35561,73
C00834=-3303,61290,2519,-938,-35561,73
C00835=-3264,61287,2516,-943,-35560,57
C00836=-3264,61287,3916,-943,-35560,57
C00837=-2723,61255,3879,-1015,-35544,-160
C00838=-2723,61255,2479,-1015,-35544,-160
C00839=-2681,61252,2476,-1020,-35543,-177
C00840=-2681,61252,3876,-1020,-35543,-177
C00841=-2460,61239,3860,-1049,-35536,-266
C00842=-2460,61239,2460,-1049,-35536,-266
C00843=-2417,61237,2457,-1055,-35535,-283
C00844=-2417,61237,3857,-1055,-35535,-283
C00845=-2298,61230,3849,-1071,-35531,-331
C00846=-2298,61230,2449,-1071,-35531,-331
C00847=-2252,61227,2446,-1077,-35530,-349
C00848=-2252,61227,3846,-1077,-35530,-349
C00849=-2098,61218,3835,-1097,-35525,-411
C00850=-2098,61218,2435,-1097,-35525,-411
C00851=-2055,61215,2432,-1103,-35524,-428
C00852=-2055,61215,3832,-1103,-35524,-428
C00853=-1996,61212,3828,-1111,-35522,-452
C00854=-1996,61212,2428,-1111,-35522,-452
C00855=-1957,61209,2425,-1116,-35521,-468
C00856=-1957,61209,3825,-1116,-35521,-468
C00857=-1827,61202,3816,-1133,-35517,-520
C00858=-1827,61202,2416,-1133,-35517,-520
C00859=-1781,61199,2413,-1139,-35516,-538
C00860=-1781,61199,3813,-1139,-35516,-538
C00861=-1514,61183,3794,-1174,-35508,-645
C00862=-1514,61183,2394,-1174,-35508,-645
C00863=-1462,61180,2391,-1181,-35506,-667
C00864=-1462,61180,3791,-1181,-35506,-667
C00865=-527,61124,3726,-1305,-35478,-1042
C00866=-527,61124,2326,-1305,-35478,-1042
C00867=-485,61121,2323,-1310,-35477,-1059
C00868=-485,61121,3723,-1310,-35477,-1059
C00869=-453,61120,3721,-1315,-35476,-1072
C00870=-453,61120,2321,-1315,-35476,-1072
C00871=-407,61117,2317,-1321,-35475,-1090
C00872=-407,61117,3717,-1321,-35475,-1090
C00873=-214,61105,3704,-1346,-35469,-1168
C00874=-214,61105,2304,-1346,-35469,-1168
C00875=-179,61103,2301,-1351,-35468,-1182
C00876=-179,61103,3701,-1351,-35468,-1182
C00877=-67,61097,3694,-1366,-35465,-1227
C00878=-67,61097,2294,-1366,-35465,-1227
C00879=-14,61093,2290,-1373,-35463,-1248
C00880=-14,61093,3690,-1373,-35463,-1248
C00881=194,61081,3676,-1400,-35457,-1331
C00882=194,61081,2276,-1400,-35457,-1331
C00883=232,61079,2273,-1405,-35456,-1347
C00884=232,61079,3673,-1405,-35456,-1347
C00885=-5426,61372,4000,-658,-35598,926
C00886=-5426,61372,2600,-658,-35598,926
C00887=-5377,61369,2596,-665,-35596,906
C00888=-5377,61369,3996,-665,-35596,906
C00889=-4962,61344,3967,-720,-35584,740
C00890=-4962,61344,2567,-720,-35584,740
C00891=-4861,61338,2560,-733,-35581,699
C00892=-4861,61338,3960,-733,-35581,699
C00893=-3982,61286,3899,-849,-35555,346
C00894=-3982,61286,2499,-849,-35555,346
C00895=-3856,61278,2490,-866,-35551,295
C00896=-3856,61278,3890,-866,-35551,295
C00897=-3290,61244,3851,-941,-35534,68
C00898=-3290,61244,2451,-941,-35534,68
C00899=-3248,61242,2448,-946,-35533,51
C00900=-3248,61242,3848,-946,-35533,51
C00901=-2706,61210,3810,-1018,-35516,-166
C00902=-2706,61210,2410,-1018,-35516,-166
C00903=-2664,61207,2407,-1023,-35515,-183
C00904=-2664,61207,3807,-1023,-35515,-183
C00905=-2474,61196,3794,-1048,-35509,-259
C00906=-2474,61196,2394,-1048,-35509,-259
C00907=-2432,61193,2391,-1054,-35508,-276
C00908=-2432,61193,3791,-1054,-35508,-276
C00909=-2281,61184,3781,-1074,-35504,-337
C00910=-2281,61184,2381,-1074,-35504,-337
C00911=-2218,61181,2376,-1082,-35502,-362
C00912=-2218,61181,3776,-1082,-35502,-362
C00913=-2127,61175,3770,-1094,-35499,-399
C00914=-2127,61175,2370,-1094,-35499,-399
C00915=-2070,61172,2366,-1102,-35497,-422
C00916=-2070,61172,3766,-1102,-35497,-422
C00917=-1986,61167,3760,-1113,-35495,-455
C00918=-1986,61167,2360,-1113,-35495,-455
C00919=-1940,61164,2357,-1119,-35493,-474
C00920=-1940,61164,3757,-1119,-35493,-474
C00921=-1824,61157,3749,-1134,-35490,-520
C00922=-1824,61157,2349,-1134,-35490,-520
C00923=-1775,61154,2346,-1141,-35489,-540
C00924=-1775,61154,3746,-1141,-35489,-540
C00925=-1515,61139,3727,-1175,-35481,-645
C00926=-1515,61139,2327,-1175,-35481,-645
C00927=-1459,61135,2324,-1182,-35479,-667
C00928=-1459,61135,3724,-1182,-35479,-667
C00929=-517,61079,3658,-1307,-35451,-1045
C00930=-517,61079,2258,-1307,-35451,-1045
C00931=-478,61077,2255,-1312,-35450,-1061
C00932=-478,61077,3655,-1312,-35450,-1061
C00933=-436,61075,3652,-1317,-35448,-1078
C00934=-436,61075,2252,-1317,-35448,-1078
C00935=-380,61071,2248,-1325,-35447,-1100
C00936=-380,61071,3648,-1325,-35447,-1100
C00937=-229,61062,3638,-1345,-35442,-1161
C00938=-229,61062,2238,-1345,-35442,-1161
C00939=-187,61060,2235,-1350,-35441,-1178
C00940=-187,61060,3635,-1350,-35441,-1178
C00941=-46,61051,3625,-1369,-35437,-1234
C00942=-46,61051,2225,-1369,-35437,-1234
C00943=24,61047,2220,-1378,-35435,-1263
C00944=24,61047,3620,-1378,-35435,-1263
C00945=182,61038,3609,-1399,-35430,-1326
C00946=182,61038,2209,-1399,-35430,-1326
C00947=221,61035,2207,-1404,-35429,-1342
C00948=221,61035,3607,-1404,-35429,-1342
C00949=-5434,61328,3933,-658,-35571,930
C00950=-5434,61328,2533,-658,-35571,930
C00951=-5389,61325,2530,-664,-35570,911
C00952=-5389,61325,3930,-664,-35570,911
C00953=-4967,61300,3901,-720,-35557,742
C00954=-4967,61300,2501,-720,-35557,742
C00955=-4851,61293,2493,-735,-35554,695
C00956=-4851,61293,3893,-735,-35554,695
C00957=-4004,61243,3834,-847,-35528,355
C00958=-4004,61243,2434,-847,-35528,355
C00959=-3842,61233,2422,-868,-35523,290
C00960=-3842,61233,3822,-868,-35523,290
C00961=-3280,61200,3783,-943,-35507,65
C00962=-3280,61200,2383,-943,-35507,65
C00963=-3231,61197,2380,-949,-35505,45
C00964=-3231,61197,3780,-949,-35505,45
C00965=-2686,61164,3742,-1021,-35489,-174
C00966=-2686,61164,2342,-1021,-35489,-174
C00967=-2637,61161,2338,-1027,-35487,-194
C00968=-2637,61161,3738,-1027,-35487,-194
C00969=-2503,61153,3729,-1045,-35483,-247
C00970=-2503,61153,2329,-1045,-35483,-247
C00971=-2447,61150,2325,-1053,-35482,-270
C00972=-2447,61150,3725,-1053,-35482,-270
C00973=-2229,61137,3710,-1081,-35475,-357
C00974=-2229,61137,2310,-1081,-35475,-357
C00975=-2099,61129,2301,-1099,-35471,-409
C00976=-2099,61129,3701,-1099,-35471,-409
C00977=-1980,61122,3693,-1114,-35468,-457
C00978=-1980,61122,2293,-1114,-35468,-457
C00979=-1924,61119,2289,-1122,-35466,-480
C00980=-1924,61119,3689,-1122,-35466,-480
C00981=-1822,61113,3682,-1135,-35463,-521
C00982=-1822,61113,2282,-1135,-35463,-521
C00983=-1769,61110,2278,-1142,-35461,-542
C00984=-1769,61110,3678,-1142,-35461,-542
C00985=-1502,61094,3659,-1177,-35453,-649
C00986=-1502,61094,2259,-1177,-35453,-649
C00987=-1467,61092,2257,-1182,-35452,-663
C00988=-1467,61092,3657,-1182,-35452,-663
C00989=-511,61035,3591,-1308,-35424,-1047
C00990=-511,61035,2191,-1308,-35424,-1047
C00991=-469,61032,2188,-1314,-35422,-1064
C00992=-469,61032,3588,-1314,-35422,-1064
C00993=-412,61029,3584,-1321,-35421,-1087
C00994=-412,61029,2184,-1321,-35421,-1087
C00995=-331,61024,2178,-1332,-35418,-1119
C00996=-331,61024,3578,-1332,-35418,-1119
C00997=-261,61020,3573,-1341,-35416,-1147
C00998=-261,61020,2173,-1341,-35416,-1147
C00999=-198,61016,2169,-1350,-35414,-1173
C01000=-198,61016,3569,-1350,-35414,-1173
C01001=-12,61005,3556,-1374,-35409,-1248
C01002=-12,61005,2156,-1374,-35409,-1248
C01003=73,61000,2150,-1385,-35406,-1281
C01004=73,61000,3550,-1385,-35406,-1281
C01005=154,60995,3544,-1396,-35404,-1314
C01006=154,60995,2144,-1396,-35404,-1314
C01007=206,60992,2141,-1403,-35402,-1335
C01008=206,60992,3541,-1403,-35402,-1335
C01009=-5442,61284,3867,-657,-35544,933
C01010=-5442,61284,2467,-657,-35544,933
C01011=-5400,61281,2464,-663,-35543,917
C01012=-5400,61281,3864,-663,-35543,917
C01013=-4978,61256,3834,-719,-35531,747
C01014=-4978,61256,2434,-719,-35531,747
C01015=-4820,61247,2423,-740,-35526,684
C01016=-4820,61247,3823,-740,-35526,684
C01017=-4008,61199,3767,-847,-35501,358
C01018=-4008,61199,2367,-847,-35501,358
C01019=-3826,61188,2354,-871,-35496,284
C01020=-3826,61188,3754,-871,-35496,284
C01021=-3267,61154,3715,-945,-35479,60
C01022=-3267,61154,2315,-945,-35479,60
C01023=-3214,61151,2312,-952,-35478,39
C01024=-3214,61151,3712,-952,-35478,39
C01025=-2659,61118,3673,-1025,-35461,-184
C01026=-2659,61118,2273,-1025,-35461,-184
C01027=-2473,61107,2260,-1050,-35455,-259
C01028=-2473,61107,3660,-1050,-35455,-259
C01029=-1815,61068,3614,-1137,-35436,-523
C01030=-1815,61068,2214,-1137,-35436,-523
C01031=-1770,61066,2211,-1143,-35434,-541
C01032=-1770,61066,3611,-1143,-35434,-541
C01033=-508,60991,3523,-1310,-35396,-1048
C01034=-508,60991,2123,-1310,-35396,-1048
C01035=-466,60988,2120,-1315,-35395,-1065
C01036=-466,60988,3520,-1315,-35395,-1065
C01037=-374,60983,3514,-1327,-35392,-1101
C01038=-374,60983,2114,-1327,-35392,-1101
C01039=-230,60974,2104,-1346,-35388,-1159
C01040=-230,60974,3504,-1346,-35388,-1159
C01041=37,60958,3485,-1382,-35380,-1266
C01042=37,60958,2085,-1382,-35380,-1266
C01043=184,60950,2075,-1401,-35376,-1326
C01044=184,60950,3475,-1401,-35376,-1326
C01045=-5450,61240,3800,-657,-35518,937
C01046=-5450,61240,2400,-657,-35518,937
C01047=-5408,61237,2397,-663,-35516,920
C01048=-5408,61237,3797,-663,-35516,920
C01049=-4983,61212,3768,-719,-35504,750
C01050=-4983,61212,2368,-719,-35504,750
C01051=-4800,61201,2355,-743,-35498,676
C01052=-4800,61201,3755,-743,-35498,676
C01053=-4016,61155,3700,-847,-35475,361
C01054=-4016,61155,2300,-847,-35475,361
C01055=-3823,61143,2287,-872,-35469,284
C01056=-3823,61143,3687,-872,-35469,284
C01057=-3250,61109,3647,-948,-35452,54
C01058=-3250,61109,2247,-948,-35452,54
C01059=-3197,61106,2243,-955,-35450,33
C01060=-3197,61106,3643,-955,-35450,33
C01061=-2610,61071,3603,-1032,-35432,-203
C01062=-2610,61071,2203,-1032,-35432,-203
C01063=-2526,61066,2197,-1044,-35430,-237
C01064=-2526,61066,3597,-1044,-35430,-237
C01065=-505,60946,3456,-1311,-35369,-1048
C01066=-505,60946,2056,-1311,-35369,-1048
C01067=-463,60944,2053,-1316,-35368,-1065
C01068=-463,60944,3453,-1316,-35368,-1065
C01069=-5459,61196,3734,-657,-35491,941
C01070=-5459,61196,2334,-657,-35491,941
C01071=-5409,61193,2330,-663,-35490,921
C01072=-5409,61193,3730,-663,-35490,921
C01073=-4991,61168,3701,-718,-35477,753
C01074=-4991,61168,2301,-718,-35477,753
C01075=-4794,61156,2287,-744,-35471,674
C01076=-4794,61156,3687,-744,-35471,674
C01077=-4021,61110,3634,-847,-35448,364
C01078=-4021,61110,2234,-847,-35448,364
C01079=-3813,61098,2219,-874,-35442,281
C01080=-3813,61098,3619,-874,-35442,281
C01081=-3233,61064,3579,-951,-35424,48
C01082=-3233,61064,2179,-951,-35424,48
C01083=-3188,61061,2176,-957,-35423,29
C01084=-3188,61061,3576,-957,-35423,29
C01085=-509,60903,3389,-1311,-35342,-1046
C01086=-509,60903,1989,-1311,-35342,-1046
C01087=-471,60900,1987,-1316,-35341,-1061
C01088=-471,60900,3387,-1316,-35341,-1061
C01089=-5467,61152,3667,-656,-35464,945
C01090=-5467,61152,2267,-656,-35464,945
C01091=-5421,61149,2264,-662,-35463,926
C01092=-5421,61149,3664,-662,-35463,926
C01093=-4996,61124,3634,-719,-35450,756
C01094=-4996,61124,2234,-719,-35450,756
C01095=-4785,61111,2220,-746,-35444,671
C01096=-4785,61111,3620,-746,-35444,671
C01097=-4029,61067,3567,-846,-35421,368
C01098=-4029,61067,2167,-846,-35421,368
C01099=-3807,61053,2152,-876,-35414,279
C01100=-3807,61053,3552,-876,-35414,279
C01101=-3220,61019,3511,-953,-35397,43
C01102=-3220,61019,2111,-953,-35397,43
C01103=-3178,61016,2108,-959,-35395,26
C01104=-3178,61016,3508,-959,-35395,26
C01105=-939,60884,3352,-1255,-35328,-873
C01106=-939,60884,1952,-1255,-35328,-873
C01107=-918,60883,1951,-1258,-35327,-881
C01108=-918,60883,3351,-1258,-35327,-881
C01109=-514,60859,3323,-1311,-35315,-1044
C01110=-514,60859,1923,-1311,-35315,-1044
C01111=-475,60856,1920,-1316,-35314,-1059
C01112=-475,60856,3320,-1316,-35314,-1059
C01113=-5475,61107,3601,-656,-35438,948
C01114=-5475,61107,2201,-656,-35438,948
C01115=-5429,61105,2197,-662,-35436,930
C01116=-5429,61105,3597,-662,-35436,930
C01117=-5004,61080,3568,-718,-35424,759
C01118=-5004,61080,2168,-718,-35424,759
C01119=-4775,61066,2152,-748,-35417,668
C01120=-4775,61066,3552,-748,-35417,668
C01121=-4033,61022,3500,-846,-35394,370
C01122=-4033,61022,2100,-846,-35394,370
C01123=-3798,61008,2084,-878,-35387,275
C01124=-3798,61008,3484,-878,-35387,275
C01125=-3214,60974,3443,-955,-35370,41
C01126=-3214,60974,2043,-955,-35370,41
C01127=-3172,60972,2040,-960,-35368,24
C01128=-3172,60972,3440,-960,-35368,24
C01129=-922,60839,3284,-1258,-35300,-879
C01130=-922,60839,1884,-1258,-35300,-879
C01131=-904,60838,1883,-1260,-35300,-886
C01132=-904,60838,3283,-1260,-35300,-886
C01133=-521,60815,3256,-1311,-35288,-1040
C01134=-521,60815,1856,-1311,-35288,-1040
C01135=-479,60813,1853,-1316,-35287,-1057
C01136=-479,60813,3253,-1316,-35287,-1057
C01137=-5479,61063,3534,-656,-35411,951
C01138=-5479,61063,2134,-656,-35411,951
C01139=-5437,61061,2131,-661,-35410,934
C01140=-5437,61061,3531,-661,-35410,934
C01141=-5008,61035,3501,-718,-35397,762
C01142=-5008,61035,2101,-718,-35397,762
C01143=-4765,61021,2084,-750,-35389,664
C01144=-4765,61021,3484,-750,-35389,664
C01145=-4041,60978,3434,-846,-35367,374
C01146=-4041,60978,2034,-846,-35367,374
C01147=-3792,60964,2016,-879,-35360,273
C01148=-3792,60964,3416,-879,-35360,273
C01149=-3208,60929,3376,-956,-35342,39
C01150=-3208,60929,1976,-956,-35342,39
C01151=-3169,60927,1973,-961,-35341,24
C01152=-3169,60927,3373,-961,-35341,24
C01153=-909,60794,3216,-1260,-35273,-884
C01154=-909,60794,1816,-1260,-35273,-884
C01155=-888,60793,1815,-1263,-35272,-892
C01156=-888,60793,3215,-1263,-35272,-892
C01157=-536,60772,3190,-1310,-35262,-1033
C01158=-536,60772,1790,-1310,-35262,-1033
C01159=-494,60769,1787,-1315,-35260,-1050
C01160=-494,60769,3187,-1315,-35260,-1050
C01161=-5484,61019,3467,-656,-35384,953
C01162=-5484,61019,2067,-656,-35384,953
C01163=-5445,61017,2064,-661,-35383,938
C01164=-5445,61017,3464,-661,-35383,938
C01165=-5013,60991,3434,-718,-35370,764
C01166=-5013,60991,2034,-718,-35370,764
C01167=-4756,60976,2016,-752,-35362,661
C01168=-4756,60976,3416,-752,-35362,661
C01169=-4046,60934,3367,-846,-35341,376
C01170=-4046,60934,1967,-846,-35341,376
C01171=-3785,60919,1949,-881,-35333,271
C01172=-3785,60919,3349,-881,-35333,271
C01173=-3202,60885,3308,-958,-35315,37
C01174=-3202,60885,1908,-958,-35315,37
C01175=-3167,60883,1906,-962,-35314,23
C01176=-3167,60883,3306,-962,-35314,23
C01177=-888,60748,3148,-1264,-35245,-891
C01178=-888,60748,1748,-1264,-35245,-891
C01179=-864,60747,1746,-1267,-35244,-901
C01180=-864,60747,3146,-1267,-35244,-901
C01181=-551,60729,3124,-1308,-35235,-1027
C01182=-551,60729,1724,-1308,-35235,-1027
C01183=-505,60726,1721,-1314,-35233,-1045
C01184=-505,60726,3121,-1314,-35233,-1045
C01185=-5492,60975,3400,-656,-35357,957
C01186=-5492,60975,2000,-656,-35357,957
C01187=-5450,60972,1997,-661,-35356,940
C01188=-5450,60972,3397,-661,-35356,940
C01189=-5014,60947,3367,-719,-35343,765
C01190=-5014,60947,1967,-719,-35343,765
C01191=-4750,60931,1949,-754,-35335,659
C01192=-4750,60931,3349,-754,-35335,659
C01193=-4050,60890,3300,-846,-35314,378
C01194=-4050,60890,1900,-846,-35314,378
C01195=-3779,60874,1881,-882,-35306,270
C01196=-3779,60874,3281,-882,-35306,270
C01197=-3199,60840,3241,-959,-35288,37
C01198=-3199,60840,1841,-959,-35288,37
C01199=-3164,60838,1839,-963,-35287,23
C01200=-3164,60838,3239,-963,-35287,23
C01201=-872,60703,3079,-1267,-35217,-898
C01202=-872,60703,1679,-1267,-35217,-898
C01203=-840,60702,1677,-1271,-35216,-910
C01204=-840,60702,3077,-1271,-35216,-910
C01205=-566,60685,3058,-1307,-35208,-1020
C01206=-566,60685,1658,-1307,-35208,-1020
C01207=-520,60683,1655,-1313,-35207,-1039
C01208=-520,60683,3055,-1313,-35207,-1039
C01209=-5503,60931,3334,-655,-35331,962
C01210=-5503,60931,1934,-655,-35331,962
C01211=-5458,60928,1931,-661,-35330,944
C01212=-5458,60928,3331,-661,-35330,944
C01213=-5018,60903,3300,-719,-35316,767
C01214=-5018,60903,1900,-719,-35316,767
C01215=-4744,60887,1881,-755,-35308,657
C01216=-4744,60887,3281,-755,-35308,657
C01217=-4051,60846,3233,-847,-35287,379
C01218=-4051,60846,1833,-847,-35287,379
C01219=-3773,60830,1814,-884,-35278,268
C01220=-3773,60830,3214,-884,-35278,268
C01221=-3193,60796,3174,-960,-35261,35
C01222=-3193,60796,1774,-960,-35261,35
C01223=-3161,60794,1771,-965,-35260,22
C01224=-3161,60794,3171,-965,-35260,22
C01225=-851,60658,3011,-1270,-35190,-905
C01226=-851,60658,1611,-1270,-35190,-905
C01227=-812,60656,1608,-1275,-35189,-921
C01228=-812,60656,3008,-1275,-35189,-921
C01229=-587,60643,2993,-1305,-35182,-1011
C01230=-587,60643,1593,-1305,-35182,-1011
C01231=-538,60640,1589,-1312,-35180,-1031
C01232=-538,60640,2989,-1312,-35180,-1031
C01233=-5508,60887,3267,-655,-35304,964
C01234=-5508,60887,1867,-655,-35304,964
C01235=-5466,60884,1864,-660,-35303,947
C01236=-5466,60884,3264,-660,-35303,947
C01237=-5019,60858,3233,-719,-35289,768
C01238=-5019,60858,1833,-719,-35289,768
C01239=-4741,60842,1814,-756,-35281,657
C01240=-4741,60842,3214,-756,-35281,657
C01241=-4052,60802,3166,-847,-35260,380
C01242=-4052,60802,1766,-847,-35260,380
C01243=-3767,60785,1746,-885,-35251,266
C01244=-3767,60785,3146,-885,-35251,266
C01245=-3190,60751,3106,-961,-35234,34
C01246=-3190,60751,1706,-961,-35234,34
C01247=-3155,60749,1704,-966,-35233,20
C01248=-3155,60749,3104,-966,-35233,20
C01249=-827,60613,2942,-1274,-35162,-914
C01250=-827,60613,1542,-1274,-35162,-914
C01251=-785,60610,1539,-1280,-35161,-931
C01252=-785,60610,2939,-1280,-35161,-931
C01253=-620,60600,2928,-1302,-35156,-997
C01254=-620,60600,1528,-1302,-35156,-997
C01255=-560,60597,1524,-1309,-35154,-1021
C01256=-560,60597,2924,-1309,-35154,-1021
C01257=-5516,60843,3201,-654,-35277,968
C01258=-5516,60843,1801,-654,-35277,968
C01259=-5474,60840,1798,-660,-35276,951
C01260=-5474,60840,3198,-660,-35276,951
C01261=-5020,60814,3166,-720,-35262,769
C01262=-5020,60814,1766,-720,-35262,769
C01263=-4732,60797,1746,-758,-35254,653
C01264=-4732,60797,3146,-758,-35254,653
C01265=-4053,60757,3099,-848,-35233,381
C01266=-4053,60757,1699,-848,-35233,381
C01267=-3765,60740,1679,-886,-35224,265
C01268=-3765,60740,3079,-886,-35224,265
C01269=-3191,60707,3039,-962,-35207,35
C01270=-3191,60707,1639,-962,-35207,35
C01271=-3153,60705,1637,-967,-35206,20
C01272=-3153,60705,3037,-967,-35206,20
C01273=-796,60567,2873,-1279,-35134,-926
C01274=-796,60567,1473,-1279,-35134,-926
C01275=-733,60563,1469,-1287,-35132,-951
C01276=-733,60563,2869,-1287,-35132,-951
C01277=-659,60559,2864,-1297,-35130,-981
C01278=-659,60559,1464,-1297,-35130,-981
C01279=-592,60555,1459,-1306,-35128,-1008
C01280=-592,60555,2859,-1306,-35128,-1008
C01281=-5520,60799,3134,-654,-35251,970
C01282=-5520,60799,1734,-654,-35251,970
C01283=-5478,60796,1731,-660,-35249,953
C01284=-5478,60796,3131,-660,-35249,953
C01285=-5021,60769,3099,-720,-35235,770
C01286=-5021,60769,1699,-720,-35235,770
C01287=-4733,60753,1679,-759,-35227,654
C01288=-4733,60753,3079,-759,-35227,654
C01289=-4054,60713,3032,-849,-35206,382
C01290=-4054,60713,1632,-849,-35206,382
C01291=-3762,60696,1612,-887,-35197,265
C01292=-3762,60696,3012,-887,-35197,265
C01293=-3185,60662,2972,-964,-35180,33
C01294=-3185,60662,1572,-964,-35180,33
C01295=-3146,60660,1569,-969,-35178,18
C01296=-3146,60660,2969,-969,-35178,18
C01297=-748,60520,2803,-1286,-35105,-945
C01298=-748,60520,1403,-1286,-35105,-945
C01299=-635,60513,1395,-1301,-35102,-990
C01300=-635,60513,2795,-1301,-35102,-990
C01301=1510,60388,2646,-1585,-35036,-1851
C01302=1510,60388,1246,-1585,-35036,-1851
C01303=1644,60380,1237,-1603,-35032,-1904
C01304=1644,60380,2637,-1603,-35032,-1904
C01305=-5525,60754,3067,-654,-35224,973
C01306=-5525,60754,1667,-654,-35224,973
C01307=-5479,60752,1664,-660,-35223,954
C01308=-5479,60752,3064,-660,-35223,954
C01309=-5018,60725,3032,-721,-35208,770
C01310=-5018,60725,1632,-721,-35208,770
C01311=-4727,60708,1612,-760,-35200,652
C01312=-4727,60708,3012,-760,-35200,652
C01313=-4044,60668,2965,-850,-35179,379
C01314=-4044,60668,1565,-850,-35179,379
C01315=-3763,60651,1545,-888,-35170,266
C01316=-3763,60651,2945,-888,-35170,266
C01317=-3182,60618,2905,-965,-35152,33
C01318=-3182,60618,1505,-965,-35152,33
C01319=-3144,60615,1502,-970,-35151,17
C01320=-3144,60615,2902,-970,-35151,17
C01321=1432,60348,2585,-1576,-35012,-1819
C01322=1432,60348,1185,-1576,-35012,-1819
C01323=1548,60342,1176,-1591,-35008,-1865
C01324=1548,60342,2576,-1591,-35008,-1865
C01325=1590,60339,2574,-1596,-35007,-1882
C01326=1590,60339,1174,-1596,-35007,-1882
C01327=1671,60334,1168,-1607,-35004,-1915
C01328=1671,60334,2568,-1607,-35004,-1915
C01329=-5533,60710,3001,-654,-35197,976
C01330=-5533,60710,1601,-654,-35197,976
C01331=-5484,60707,1597,-661,-35196,957
C01332=-5484,60707,2997,-661,-35196,957
C01333=-5016,60680,2965,-722,-35181,769
C01334=-5016,60680,1565,-722,-35181,769
C01335=-4724,60663,1545,-761,-35173,652
C01336=-4724,60663,2945,-761,-35173,652
C01337=-4038,60623,2897,-852,-35152,377
C01338=-4038,60623,1497,-852,-35152,377
C01339=-3760,60607,1478,-889,-35143,265
C01340=-3760,60607,2878,-889,-35143,265
C01341=-3176,60573,2837,-966,-35125,31
C01342=-3176,60573,1437,-966,-35125,31
C01343=-3141,60571,1435,-971,-35124,17
C01344=-3141,60571,2835,-971,-35124,17
C01345=-222,60401,2632,-1357,-35035,-1155
C01346=-222,60401,1232,-1357,-35035,-1155
C01347=-172,60398,1229,-1364,-35033,-1174
C01348=-172,60398,2629,-1364,-35033,-1174
C01349=17,60387,2616,-1389,-35028,-1251
C01350=17,60387,1216,-1389,-35028,-1251
C01351=46,60385,1214,-1393,-35027,-1262
C01352=46,60385,2614,-1393,-35027,-1262
C01353=1393,60307,2520,-1571,-34986,-1802
C01354=1393,60307,1120,-1571,-34986,-1802
C01355=1467,60302,1115,-1581,-34983,-1832
C01356=1467,60302,2515,-1581,-34983,-1832
C01357=1635,60293,2503,-1603,-34978,-1900
C01358=1635,60293,1103,-1603,-34978,-1900
C01359=1681,60290,1100,-1609,-34977,-1918
C01360=1681,60290,2500,-1609,-34977,-1918
C01361=-5531,60666,2933,-655,-35170,976
C01362=-5531,60666,1533,-655,-35170,976
C01363=-5481,60663,1530,-662,-35169,956
C01364=-5481,60663,2930,-662,-35169,956
C01365=-5010,60635,2897,-724,-35154,767
C01366=-5010,60635,1497,-724,-35154,767
C01367=-4725,60619,1478,-762,-35146,653
C01368=-4725,60619,2878,-762,-35146,653
C01369=-4021,60578,2829,-855,-35124,371
C01370=-4021,60578,1429,-855,-35124,371
C01371=-3761,60563,1411,-889,-35116,266
C01372=-3761,60563,2811,-889,-35116,266
C01373=-3174,60528,2770,-967,-35098,30
C01374=-3174,60528,1370,-967,-35098,30
C01375=-3131,60526,1367,-973,-35097,13
C01376=-3131,60526,2767,-973,-35097,13
C01377=-2621,60496,2732,-1040,-35081,-191
C01378=-2621,60496,1332,-1040,-35081,-191
C01379=-2583,60494,1329,-1045,-35080,-207
C01380=-2583,60494,2729,-1045,-35080,-207
C01381=-222,60357,2565,-1358,-35008,-1154
C01382=-222,60357,1165,-1358,-35008,-1154
C01383=-173,60354,1162,-1365,-35006,-1174
C01384=-173,60354,2562,-1365,-35006,-1174
C01385=13,60343,2549,-1389,-35001,-1248
C01386=13,60343,1149,-1389,-35001,-1248
C01387=55,60341,1146,-1395,-34999,-1265
C01388=55,60341,2546,-1395,-34999,-1265
C01389=1368,60264,2455,-1569,-34959,-1792
C01390=1368,60264,1055,-1569,-34959,-1792
C01391=1424,60261,1051,-1576,-34957,-1814
C01392=1424,60261,2451,-1576,-34957,-1814
C01393=1645,60248,2436,-1605,-34951,-1903
C01394=1645,60248,1036,-1605,-34951,-1903
C01395=1688,60246,1033,-1611,-34949,-1920
C01396=1688,60246,2433,-1611,-34949,-1920
C01397=-5528,60621,2866,-656,-35143,976
C01398=-5528,60621,1466,-656,-35143,976
C01399=-5482,60618,1463,-662,-35142,957
C01400=-5482,60618,2863,-662,-35142,957
C01401=-5004,60590,2830,-725,-35127,765
C01402=-5004,60590,1430,-725,-35127,765
C01403=-4726,60574,1411,-762,-35119,654
C01404=-4726,60574,2811,-762,-35119,654
C01405=-4012,60533,2761,-857,-35097,367
C01406=-4012,60533,1361,-857,-35097,367
C01407=-3762,60518,1344,-890,-35089,267
C01408=-3762,60518,2744,-890,-35089,267
C01409=-3168,60484,2703,-969,-35071,28
C01410=-3168,60484,1303,-969,-35071,28
C01411=-3129,60482,1300,-974,-35070,13
C01412=-3129,60482,2700,-974,-35070,13
C01413=-2619,60452,2664,-1041,-35054,-192
C01414=-2619,60452,1264,-1041,-35054,-192
C01415=-2573,60449,1261,-1047,-35053,-210
C01416=-2573,60449,2661,-1047,-35053,-210
C01417=-220,60313,2498,-1359,-34981,-1154
C01418=-220,60313,1098,-1359,-34981,-1154
C01419=-174,60310,1095,-1365,-34979,-1173
C01420=-174,60310,2495,-1365,-34979,-1173
C01421=23,60298,2481,-1391,-34973,-1252
C01422=23,60298,1081,-1391,-34973,-1252
C01423=62,60296,1079,-1396,-34972,-1267
C01424=62,60296,2479,-1396,-34972,-1267
C01425=1363,60221,2388,-1569,-34932,-1789
C01426=1363,60221,988,-1569,-34932,-1789
C01427=1402,60218,986,-1574,-34931,-1805
C01428=1402,60218,2386,-1574,-34931,-1805
C01429=1645,60204,2369,-1606,-34923,-1902
C01430=1645,60204,969,-1606,-34923,-1902
C01431=1687,60202,966,-1612,-34922,-1919
C01432=1687,60202,2366,-1612,-34922,-1919
C01433=-5526,60576,2799,-657,-35116,975
C01434=-5526,60576,1399,-657,-35116,975
C01435=-5483,60574,1396,-663,-35115,958
C01436=-5483,60574,2796,-663,-35115,958
C01437=-4991,60545,2762,-728,-35100,761
C01438=-4991,60545,1362,-728,-35100,761
C01439=-4741,60531,1345,-761,-35092,660
C01440=-4741,60531,2745,-761,-35092,660
C01441=-4002,60488,2693,-859,-35070,364
C01442=-4002,60488,1293,-859,-35070,364
C01443=-3763,60474,1277,-890,-35062,268
C01444=-3763,60474,2677,-890,-35062,268
C01445=-3165,60439,2635,-970,-35044,28
C01446=-3165,60439,1235,-970,-35044,28
C01447=-3130,60437,1233,-974,-35043,14
C01448=-3130,60437,2633,-974,-35043,14
C01449=-2613,60407,2597,-1043,-35027,-194
C01450=-2613,60407,1197,-1043,-35027,-194
C01451=-2567,60405,1194,-1049,-35025,-212
C01452=-2567,60405,2594,-1049,-35025,-212
C01453=-213,60268,2431,-1361,-34953,-1156
C01454=-213,60268,1031,-1361,-34953,-1156
C01455=-167,60265,1027,-1367,-34952,-1175
C01456=-167,60265,2427,-1367,-34952,-1175
C01457=33,60254,2414,-1393,-34946,-1255
C01458=33,60254,1014,-1393,-34946,-1255
C01459=75,60251,1011,-1399,-34944,-1272
C01460=75,60251,2411,-1399,-34944,-1272
C01461=571,60223,2376,-1465,-34929,-1471
C01462=571,60223,976,-1465,-34929,-1471
C01463=610,60220,974,-1470,-34928,-1486
C01464=610,60220,2374,-1470,-34928,-1486
C01465=1644,60160,2302,-1607,-34896,-1901
C01466=1644,60160,902,-1607,-34896,-1901
C01467=1687,60158,899,-1612,-34895,-1918
C01468=1687,60158,2299,-1612,-34895,-1918
C01469=-5527,60532,2732,-657,-35089,976
C01470=-5527,60532,1332,-657,-35089,976
C01471=-5477,60529,1329,-664,-35088,956
C01472=-5477,60529,2729,-664,-35088,956
C01473=-4978,60500,2694,-730,-35073,756
C01474=-4978,60500,1294,-730,-35073,756
C01475=-4749,60487,1278,-761,-35065,664
C01476=-4749,60487,2678,-761,-35065,664
C01477=-3993,60443,2626,-861,-35042,361
C01478=-3993,60443,1226,-861,-35042,361
C01479=-3767,60430,1210,-891,-35035,270
C01480=-3767,60430,2610,-891,-35035,270
C01481=-3166,60395,2568,-970,-35017,29
C01482=-3166,60395,1168,-970,-35017,29
C01483=-3127,60393,1166,-975,-35016,13
C01484=-3127,60393,2566,-975,-35016,13
C01485=-2603,60362,2529,-1045,-35000,-197
C01486=-2603,60362,1129,-1045,-35000,-197
C01487=-2557,60360,1126,-1051,-34998,-215
C01488=-2557,60360,2526,-1051,-34998,-215
C01489=-207,60224,2363,-1362,-34926,-1158
C01490=-207,60224,963,-1362,-34926,-1158
C01491=-165,60221,960,-1368,-34925,-1175
C01492=-165,60221,2360,-1368,-34925,-1175
C01493=43,60209,2346,-1395,-34918,-1258
C01494=43,60209,946,-1395,-34918,-1258
C01495=82,60207,943,-1401,-34917,-1274
C01496=82,60207,2343,-1401,-34917,-1274
C01497=1637,60117,2235,-1607,-34869,-1898
C01498=1637,60117,835,-1607,-34869,-1898
C01499=1679,60114,832,-1612,-34868,-1915
C01500=1679,60114,2232,-1612,-34868,-1915
C01501=-5524,60487,2665,-658,-35062,975
C01502=-5524,60487,1265,-658,-35062,975
C01503=-5475,60484,1261,-665,-35061,956
C01504=-5475,60484,2661,-665,-35061,956
C01505=-4961,60455,2626,-733,-35045,750
C01506=-4961,60455,1226,-733,-35045,750
C01507=-4753,60443,1211,-761,-35039,666
C01508=-4753,60443,2611,-761,-35039,666
C01509=-3976,60398,2557,-864,-35015,354
C01510=-3976,60398,1157,-864,-35015,354
C01511=-3775,60386,1143,-890,-35009,274
C01512=-3775,60386,2543,-890,-35009,274
C01513=-3167,60351,2501,-971,-34990,30
C01514=-3167,60351,1101,-971,-34990,30
C01515=-3124,60348,1098,-976,-34989,13
C01516=-3124,60348,2498,-976,-34989,13
C01517=-2597,60318,2462,-1046,-34972,-199
C01518=-2597,60318,1062,-1046,-34972,-199
C01519=-2547,60315,1058,-1053,-34971,-219
C01520=-2547,60315,2458,-1053,-34971,-219
C01521=-201,60179,2296,-1364,-34899,-1160
C01522=-201,60179,896,-1364,-34899,-1160
C01523=-162,60177,893,-1369,-34897,-1176
C01524=-162,60177,2293,-1369,-34897,-1176
C01525=53,60165,2278,-1398,-34891,-1262
C01526=53,60165,878,-1398,-34891,-1262
C01527=95,60162,875,-1403,-34889,-1279
C01528=95,60162,2275,-1403,-34889,-1279
C01529=1633,60073,2169,-1607,-34842,-1895
C01530=1633,60073,769,-1607,-34842,-1895
C01531=1671,60071,766,-1612,-34841,-1911
C01532=1671,60071,2166,-1612,-34841,-1911
C01533=-5518,60442,2597,-660,-35035,974
C01534=-5518,60442,1197,-660,-35035,974
C01535=-5472,60440,1194,-666,-35034,955
C01536=-5472,60440,2594,-666,-35034,955
C01537=-4934,60409,2557,-737,-35017,739
C01538=-4934,60409,1157,-737,-35017,739
C01539=-4765,60399,1145,-760,-35012,672
C01540=-4765,60399,2545,-760,-35012,672
C01541=-3959,60352,2489,-867,-34987,348
C01542=-3959,60352,1089,-867,-34987,348
C01543=-3787,60342,1077,-889,-34982,279
C01544=-3787,60342,2477,-889,-34982,279
C01545=-3171,60307,2435,-971,-34963,32
C01546=-3171,60307,1035,-971,-34963,32
C01547=-3132,60304,1032,-976,-34962,17
C01548=-3132,60304,2432,-976,-34962,17
C01549=-2583,60273,2394,-1049,-34945,-204
C01550=-2583,60273,994,-1049,-34945,-204
C01551=-2541,60270,991,-1054,-34944,-221
C01552=-2541,60270,2391,-1054,-34944,-221
C01553=-2084,60244,2359,-1115,-34929,-404
C01554=-2084,60244,959,-1115,-34929,-404
C01555=-1992,60239,953,-1127,-34927,-441
C01556=-1992,60239,2353,-1127,-34927,-441
C01557=-1788,60227,2339,-1154,-34920,-523
C01558=-1788,60227,939,-1154,-34920,-523
C01559=-1714,60223,934,-1164,-34918,-552
C01560=-1714,60223,2334,-1164,-34918,-552
C01561=-1327,60200,2307,-1215,-34906,-707
C01562=-1327,60200,907,-1215,-34906,-707
C01563=-1204,60193,898,-1232,-34902,-757
C01564=-1204,60193,2298,-1232,-34902,-757
C01565=-926,60177,2279,-1269,-34894,-868
C01566=-926,60177,879,-1269,-34894,-868
C01567=-782,60169,869,-1288,-34889,-926
C01568=-782,60169,2269,-1288,-34889,-926
C01569=-194,60135,2228,-1366,-34871,-1162
C01570=-194,60135,828,-1366,-34871,-1162
C01571=-155,60133,826,-1371,-34870,-1177
C01572=-155,60133,2226,-1371,-34870,-1177
C01573=66,60120,2210,-1400,-34863,-1266
C01574=66,60120,810,-1400,-34863,-1266
C01575=105,60118,808,-1405,-34862,-1282
C01576=105,60118,2208,-1405,-34862,-1282
C01577=872,60073,2154,-1507,-34838,-1590
C01578=872,60073,754,-1507,-34838,-1590
C01579=956,60068,749,-1518,-34836,-1624
C01580=956,60068,2149,-1518,-34836,-1624
C01581=1618,60030,2103,-1606,-34815,-1889
C01582=1618,60030,703,-1606,-34815,-1889
C01583=1660,60028,700,-1611,-34814,-1906
C01584=1660,60028,2100,-1611,-34814,-1906
C01585=-5516,60398,2530,-661,-35008,973
C01586=-5516,60398,1130,-661,-35008,973
C01587=-5470,60395,1127,-667,-35007,955
C01588=-5470,60395,2527,-667,-35007,955
C01589=-4872,60360,2485,-746,-34988,715
C01590=-4872,60360,1085,-746,-34988,715
C01591=-4805,60357,1081,-755,-34986,688
C01592=-4805,60357,2481,-755,-34986,688
C01593=-3943,60307,2421,-869,-34960,342
C01594=-3943,60307,1021,-869,-34960,342
C01595=-3798,60299,1011,-889,-34955,284
C01596=-3798,60299,2411,-889,-34955,284
C01597=-3175,60263,2368,-971,-34936,34
C01598=-3175,60263,968,-971,-34936,34
C01599=-3137,60260,965,-976,-34935,19
C01600=-3137,60260,2365,-976,-34935,19
C01601=-2574,60228,2326,-1051,-34917,-207
C01602=-2574,60228,926,-1051,-34917,-207
C01603=-2531,60226,923,-1056,-34916,-224
C01604=-2531,60226,2323,-1056,-34916,-224
C01605=-2109,60201,2294,-1112,-34903,-393
C01606=-2109,60201,894,-1112,-34903,-393
C01607=-2060,60198,891,-1119,-34902,-413
C01608=-2060,60198,2291,-1119,-34902,-413
C01609=-1997,60195,2286,-1127,-34900,-438
C01610=-1997,60195,886,-1127,-34900,-438
C01611=-1975,60193,885,-1130,-34899,-447
C01612=-1975,60193,2285,-1130,-34899,-447
C01613=-1831,60185,2275,-1149,-34895,-505
C01614=-1831,60185,875,-1149,-34895,-505
C01615=-1690,60177,865,-1168,-34890,-561
C01616=-1690,60177,2265,-1168,-34890,-561
C01617=-1381,60159,2243,-1209,-34881,-685
C01618=-1381,60159,843,-1209,-34881,-685
C01619=-1268,60153,836,-1224,-34877,-731
C01620=-1268,60153,2236,-1224,-34877,-731
C01621=-1236,60151,2233,-1228,-34876,-743
C01622=-1236,60151,833,-1228,-34876,-743
C01623=-1177,60147,829,-1236,-34874,-767
C01624=-1177,60147,2229,-1236,-34874,-767
C01625=-962,60135,2214,-1265,-34868,-853
C01626=-962,60135,814,-1265,-34868,-853
C01627=-902,60132,810,-1272,-34866,-877
C01628=-902,60132,2210,-1272,-34866,-877
C01629=-797,60125,2203,-1286,-34863,-920
C01630=-797,60125,803,-1286,-34863,-920
C01631=-744,60122,799,-1293,-34861,-941
C01632=-744,60122,2199,-1293,-34861,-941
C01633=-188,60090,2161,-1367,-34844,-1164
C01634=-188,60090,761,-1367,-34844,-1164
C01635=-146,60088,758,-1373,-34843,-1181
C01636=-146,60088,2158,-1373,-34843,-1181
C01637=76,60075,2143,-1402,-34836,-1270
C01638=76,60075,743,-1402,-34836,-1270
C01639=118,60073,740,-1408,-34834,-1287
C01640=118,60073,2140,-1408,-34834,-1287
C01641=812,60033,2092,-1500,-34813,-1565
C01642=812,60033,692,-1500,-34813,-1565
C01643=1026,60020,677,-1528,-34806,-1651
C01644=1026,60020,2077,-1528,-34806,-1651
C01645=1607,59987,2037,-1605,-34788,-1884
C01646=1607,59987,637,-1605,-34788,-1884
C01647=1653,59984,633,-1611,-34787,-1902
C01648=1653,59984,2033,-1611,-34787,-1902
C01649=-5513,60353,2463,-662,-34981,973
C01650=-5513,60353,1063,-662,-34981,973
C01651=-5467,60350,1059,-668,-34980,954
C01652=-5467,60350,2459,-668,-34980,954
C01653=-3919,60261,2352,-873,-34932,333
C01654=-3919,60261,952,-873,-34932,333
C01655=-3817,60255,945,-887,-34929,292
C01656=-3817,60255,2345,-887,-34929,292
C01657=-3180,60219,2301,-971,-34909,37
C01658=-3180,60219,901,-971,-34909,37
C01659=-3141,60216,898,-976,-34908,21
C01660=-3141,60216,2298,-976,-34908,21
C01661=-2567,60183,2259,-1052,-34890,-209
C01662=-2567,60183,859,-1052,-34890,-209
C01663=-2525,60181,856,-1058,-34889,-226
C01664=-2525,60181,2256,-1058,-34889,-226
C01665=-2272,60166,2238,-1092,-34881,-327
C01666=-2272,60166,838,-1092,-34881,-327
C01667=-2226,60164,835,-1098,-34880,-346
C01668=-2226,60164,2235,-1098,-34880,-346
C01669=-2128,60158,2228,-1111,-34877,-385
C01670=-2128,60158,828,-1111,-34877,-385
C01671=-2092,60156,826,-1115,-34876,-399
C01672=-2092,60156,2226,-1115,-34876,-399
C01673=-1867,60143,2210,-1145,-34869,-490
C01674=-1867,60143,810,-1145,-34869,-490
C01675=-1800,60139,806,-1154,-34867,-517
C01676=-1800,60139,2206,-1154,-34867,-517
C01677=-1698,60133,2198,-1168,-34863,-557
C01678=-1698,60133,798,-1168,-34863,-557
C01679=-1660,60131,796,-1173,-34862,-573
C01680=-1660,60131,2196,-1173,-34862,-573
C01681=-1403,60116,2178,-1207,-34854,-676
C01682=-1403,60116,778,-1207,-34854,-676
C01683=-1343,60113,774,-1215,-34852,-700
C01684=-1343,60113,2174,-1215,-34852,-700
C01685=-1195,60104,2164,-1234,-34848,-759
C01686=-1195,60104,764,-1234,-34848,-759
C01687=-1160,60102,761,-1239,-34847,-773
C01688=-1160,60102,2161,-1239,-34847,-773
C01689=-991,60093,2149,-1261,-34841,-841
C01690=-991,60093,749,-1261,-34841,-841
C01691=-935,60089,746,-1269,-34840,-864
C01692=-935,60089,2146,-1269,-34840,-864
C01693=-766,60080,2134,-1291,-34835,-932
C01694=-766,60080,734,-1291,-34835,-932
C01695=-723,60077,731,-1297,-34833,-948
C01696=-723,60077,2131,-1297,-34833,-948
C01697=-182,60046,2093,-1369,-34816,-1166
C01698=-182,60046,693,-1369,-34816,-1166
C01699=-143,60044,691,-1374,-34815,-1181
C01700=-143,60044,2091,-1374,-34815,-1181
C01701=86,60031,2075,-1404,-34808,-1273
C01702=86,60031,675,-1404,-34808,-1273
C01703=128,60028,672,-1410,-34807,-1290
C01704=128,60028,2072,-1410,-34807,-1290
C01705=565,60003,2042,-1468,-34793,-1465
C01706=565,60003,642,-1468,-34793,-1465
C01707=603,60001,639,-1473,-34792,-1481
C01708=603,60001,2039,-1473,-34792,-1481
C01709=783,59990,2027,-1497,-34787,-1553
C01710=783,59990,627,-1497,-34787,-1553
C01711=853,59986,622,-1506,-34784,-1581
C01712=853,59986,2022,-1506,-34784,-1581
C01713=987,59979,2012,-1524,-34780,-1634
C01714=987,59979,612,-1524,-34780,-1634
C01715=1061,59974,607,-1534,-34778,-1664
C01716=1061,59974,2007,-1534,-34778,-1664
C01717=1592,59944,1971,-1604,-34762,-1877
C01718=1592,59944,571,-1604,-34762,-1877
C01719=1638,59941,567,-1610,-34760,-1896
C01720=1638,59941,1967,-1610,-34760,-1896
C01721=-5510,60308,2395,-663,-34954,972
C01722=-5510,60308,995,-663,-34954,972
C01723=-5465,60306,992,-669,-34953,954
C01724=-5465,60306,2392,-669,-34953,954
C01725=-3874,60214,2282,-880,-34904,316
C01726=-3874,60214,882,-880,-34904,316
C01727=-3839,60212,880,-885,-34903,302
C01728=-3839,60212,2280,-885,-34903,302
C01729=-3188,60175,2235,-971,-34882,41
C01730=-3188,60175,835,-971,-34882,41
C01731=-3145,60172,832,-977,-34881,24
C01732=-3145,60172,2232,-977,-34881,24
C01733=-2565,60139,2191,-1054,-34863,-209
C01734=-2565,60139,791,-1054,-34863,-209
C01735=-2523,60136,788,-1059,-34862,-226
C01736=-2523,60136,2188,-1059,-34862,-226
C01737=-2347,60126,2176,-1082,-34856,-297
C01738=-2347,60126,776,-1082,-34856,-297
C01739=-2220,60119,768,-1099,-34852,-348
C01740=-2220,60119,2168,-1099,-34852,-348
C01741=-2142,60115,2162,-1110,-34850,-379
C01742=-2142,60115,762,-1110,-34850,-379
C01743=-2111,60113,760,-1114,-34849,-391
C01744=-2111,60113,2160,-1114,-34849,-391
C01745=-1893,60100,2145,-1143,-34842,-479
C01746=-1893,60100,745,-1143,-34842,-479
C01747=-1829,60097,740,-1151,-34840,-504
C01748=-1829,60097,2140,-1151,-34840,-504
C01749=-1696,60089,2131,-1169,-34836,-558
C01750=-1696,60089,731,-1169,-34836,-558
C01751=-1646,60086,728,-1175,-34835,-578
C01752=-1646,60086,2128,-1175,-34835,-578
C01753=-1417,60073,2112,-1206,-34828,-669
C01754=-1417,60073,712,-1206,-34828,-669
C01755=-1372,60070,709,-1212,-34826,-688
C01756=-1372,60070,2109,-1212,-34826,-688
C01757=-1168,60059,2095,-1239,-34820,-770
C01758=-1168,60059,695,-1239,-34820,-770
C01759=-1150,60058,693,-1241,-34819,-777
C01760=-1150,60058,2093,-1241,-34819,-777
C01761=-1009,60049,2084,-1260,-34815,-833
C01762=-1009,60049,684,-1260,-34815,-833
C01763=-960,60047,680,-1266,-34813,-853
C01764=-960,60047,2080,-1266,-34813,-853
C01765=-752,60035,2066,-1294,-34807,-936
C01766=-752,60035,666,-1294,-34807,-936
C01767=-721,60033,664,-1298,-34806,-949
C01768=-721,60033,2064,-1298,-34806,-949
C01769=-175,60002,2026,-1370,-34789,-1168
C01770=-175,60002,626,-1370,-34789,-1168
C01771=-136,59999,623,-1376,-34788,-1183
C01772=-136,59999,2023,-1376,-34788,-1183
C01773=82,59987,2008,-1404,-34781,-1271
C01774=82,59987,608,-1404,-34781,-1271
C01775=135,59984,604,-1411,-34780,-1292
C01776=135,59984,2004,-1411,-34780,-1292
C01777=314,59973,1992,-1435,-34774,-1364
C01778=314,59973,592,-1435,-34774,-1364
C01779=370,59970,588,-1443,-34772,-1387
C01780=370,59970,1988,-1443,-34772,-1387
C01781=574,59958,1974,-1470,-34766,-1468
C01782=574,59958,574,-1470,-34766,-1468
C01783=617,59956,571,-1475,-34765,-1485
C01784=617,59956,1971,-1475,-34765,-1485
C01785=754,59948,1962,-1494,-34760,-1540
C01786=754,59948,562,-1494,-34760,-1540
C01787=814,59945,557,-1502,-34759,-1564
C01788=814,59945,1957,-1502,-34759,-1564
C01789=1025,59933,1943,-1530,-34752,-1649
C01790=1025,59933,543,-1530,-34752,-1649
C01791=1074,59930,539,-1536,-34750,-1669
C01792=1074,59930,1939,-1536,-34750,-1669
C01793=1570,59901,1905,-1602,-34735,-1868
C01794=1570,59901,505,-1602,-34735,-1868
C01795=1620,59898,502,-1608,-34734,-1888
C01796=1620,59898,1902,-1608,-34734,-1888
C01797=-5508,60264,2328,-664,-34927,972
C01798=-5508,60264,928,-664,-34927,972
C01799=-5462,60261,925,-670,-34926,953
C01800=-5462,60261,2325,-670,-34926,953
C01801=-3196,60131,2168,-971,-34856,44
C01802=-3196,60131,768,-971,-34856,44
C01803=-3150,60128,765,-977,-34854,26
C01804=-3150,60128,2165,-977,-34854,26
C01805=-2559,60094,2124,-1055,-34836,-211
C01806=-2559,60094,724,-1055,-34836,-211
C01807=-2516,60092,721,-1061,-34835,-228
C01808=-2516,60092,2121,-1061,-34835,-228
C01809=-2460,60089,2117,-1068,-34833,-251
C01810=-2460,60089,717,-1068,-34833,-251
C01811=-2309,60080,707,-1088,-34828,-311
C01812=-2309,60080,2107,-1088,-34828,-311
C01813=-2266,60078,2104,-1094,-34827,-328
C01814=-2266,60078,704,-1094,-34827,-328
C01815=-2221,60075,701,-1100,-34825,-347
C01816=-2221,60075,2101,-1100,-34825,-347
C01817=-2154,60071,2096,-1109,-34823,-374
C01818=-2154,60071,696,-1109,-34823,-374
C01819=-2126,60069,694,-1112,-34822,-385
C01820=-2126,60069,2094,-1112,-34822,-385
C01821=-1911,60057,2079,-1141,-34816,-471
C01822=-1911,60057,679,-1141,-34816,-471
C01823=-1858,60054,675,-1148,-34814,-492
C01824=-1858,60054,2075,-1148,-34814,-492
C01825=-1693,60045,2064,-1170,-34809,-558
C01826=-1693,60045,664,-1170,-34809,-558
C01827=-1633,60041,660,-1178,-34807,-582
C01828=-1633,60041,2060,-1178,-34807,-582
C01829=-1432,60030,2046,-1204,-34801,-663
C01830=-1432,60030,646,-1204,-34801,-663
C01831=-1387,60027,643,-1210,-34800,-681
C01832=-1387,60027,2043,-1210,-34800,-681
C01833=-1021,60006,2017,-1259,-34788,-828
C01834=-1021,60006,617,-1259,-34788,-828
C01835=-982,60004,615,-1264,-34787,-844
C01836=-982,60004,2015,-1264,-34787,-844
C01837=-753,59991,1999,-1295,-34780,-935
C01838=-753,59991,599,-1295,-34780,-935
C01839=-718,59989,597,-1299,-34779,-949
C01840=-718,59989,1997,-1299,-34779,-949
C01841=-172,59957,1959,-1372,-34762,-1168
C01842=-172,59957,559,-1372,-34762,-1168
C01843=-134,59955,556,-1377,-34761,-1184
C01844=-134,59955,1956,-1377,-34761,-1184
C01845=7,59947,1946,-1395,-34756,-1240
C01846=7,59947,546,-1395,-34756,-1240
C01847=63,59944,542,-1403,-34755,-1263
C01848=63,59944,1942,-1403,-34755,-1263
C01849=106,59941,1939,-1408,-34753,-1280
C01850=106,59941,539,-1408,-34753,-1280
C01851=144,59939,537,-1414,-34752,-1295
C01852=144,59939,1937,-1414,-34752,-1295
C01853=271,59932,1928,-1430,-34748,-1346
C01854=271,59932,528,-1430,-34748,-1346
C01855=412,59924,518,-1449,-34744,-1403
C01856=412,59924,1918,-1449,-34744,-1403
C01857=581,59914,1907,-1471,-34739,-1470
C01858=581,59914,507,-1471,-34739,-1470
C01859=623,59912,504,-1477,-34737,-1487
C01860=623,59912,1904,-1477,-34737,-1487
C01861=743,59905,1895,-1493,-34734,-1535
C01862=743,59905,495,-1493,-34734,-1535
C01863=789,59902,492,-1499,-34732,-1554
C01864=789,59902,1892,-1499,-34732,-1554
C01865=1049,59887,1874,-1534,-34724,-1658
C01866=1049,59887,474,-1534,-34724,-1658
C01867=1084,59885,472,-1538,-34723,-1672
C01868=1084,59885,1872,-1538,-34723,-1672
C01869=1556,59858,1839,-1601,-34708,-1861
C01870=1556,59858,439,-1601,-34708,-1861
C01871=1602,59855,436,-1607,-34707,-1880
C01872=1602,59855,1836,-1607,-34707,-1880
C01873=-5505,60219,2261,-665,-34900,971
C01874=-5505,60219,861,-665,-34900,971
C01875=-5460,60216,858,-671,-34899,953
C01876=-5460,60216,2258,-671,-34899,953
C01877=-3204,60087,2102,-970,-34829,48
C01878=-3204,60087,702,-970,-34829,48
C01879=-3168,60085,699,-975,-34828,34
C01880=-3168,60085,2099,-975,-34828,34
C01881=-2577,60051,2058,-1053,-34809,-203
C01882=-2577,60051,658,-1053,-34809,-203
C01883=-2415,60042,647,-1075,-34804,-268
C01884=-2415,60042,2047,-1075,-34804,-268
C01885=-2260,60033,2036,-1095,-34800,-330
C01886=-2260,60033,636,-1095,-34800,-330
C01887=-2214,60030,633,-1101,-34798,-349
C01888=-2214,60030,2033,-1101,-34798,-349
C01889=-2165,60027,2030,-1108,-34797,-368
C01890=-2165,60027,630,-1108,-34797,-368
C01891=-2130,60025,627,-1113,-34796,-383
C01892=-2130,60025,2027,-1113,-34796,-383
C01893=-1929,60014,2013,-1139,-34789,-463
C01894=-1929,60014,613,-1139,-34789,-463
C01895=-1877,60011,610,-1146,-34788,-484
C01896=-1877,60011,2010,-1146,-34788,-484
C01897=-1687,60000,1997,-1171,-34782,-560
C01898=-1687,60000,597,-1171,-34782,-560
C01899=-1627,59997,592,-1179,-34780,-584
C01900=-1627,59997,1992,-1179,-34780,-584
C01901=-1440,59986,1979,-1204,-34774,-659
C01902=-1440,59986,579,-1204,-34774,-659
C01903=-1401,59984,577,-1209,-34773,-675
C01904=-1401,59984,1977,-1209,-34773,-675
C01905=-1035,59963,1951,-1258,-34762,-822
C01906=-1035,59963,551,-1258,-34762,-822
C01907=-993,59960,549,-1263,-34760,-838
C01908=-993,59960,1949,-1263,-34760,-838
C01909=-775,59948,1933,-1292,-34753,-926
C01910=-775,59948,533,-1292,-34753,-926
C01911=-729,59945,530,-1298,-34752,-944
C01912=-729,59945,1930,-1298,-34752,-944
C01913=-328,59922,1902,-1352,-34740,-1105
C01914=-328,59922,502,-1352,-34740,-1105
C01915=21,59902,478,-1398,-34729,-1245
C01916=21,59902,1878,-1398,-34729,-1245
C01917=112,59897,1872,-1410,-34726,-1282
C01918=112,59897,472,-1410,-34726,-1282
C01919=151,59895,469,-1415,-34725,-1297
C01920=151,59895,1869,-1415,-34725,-1297
C01921=246,59889,1863,-1428,-34722,-1335
C01922=246,59889,463,-1428,-34722,-1335
C01923=285,59887,460,-1433,-34721,-1351
C01924=285,59887,1860,-1433,-34721,-1351
C01925=387,59881,1853,-1446,-34717,-1392
C01926=387,59881,453,-1446,-34717,-1392
C01927=439,59878,449,-1453,-34716,-1413
C01928=439,59878,1849,-1453,-34716,-1413
C01929=587,59870,1839,-1473,-34711,-1472
C01930=587,59870,439,-1473,-34711,-1472
C01931=629,59867,436,-1479,-34710,-1489
C01932=629,59867,1836,-1479,-34710,-1489
C01933=739,59861,1829,-1493,-34706,-1533
C01934=739,59861,429,-1493,-34706,-1533
C01935=781,59859,426,-1499,-34705,-1550
C01936=781,59859,1826,-1499,-34705,-1550
C01937=1534,59815,1774,-1599,-34682,-1852
C01938=1534,59815,374,-1599,-34682,-1852
C01939=1583,59813,370,-1605,-34680,-1872
C01940=1583,59813,1770,-1605,-34680,-1872
C01941=-5503,60174,2194,-666,-34873,971
C01942=-5503,60174,794,-666,-34873,971
C01943=-5457,60172,790,-672,-34872,952
C01944=-5457,60172,2190,-672,-34872,952
C01945=-3215,60043,2035,-969,-34802,53
C01946=-3215,60043,635,-969,-34802,53
C01947=-3173,60041,632,-975,-34801,36
C01948=-3173,60041,2032,-975,-34801,36
C01949=-2740,60016,2002,-1032,-34787,-137
C01950=-2740,60016,602,-1032,-34787,-137
C01951=-2507,60003,586,-1063,-34780,-231
C01952=-2507,60003,1986,-1063,-34780,-231
C01953=-2254,59988,1969,-1097,-34772,-332
C01954=-2254,59988,569,-1097,-34772,-332
C01955=-2205,59986,565,-1103,-34771,-352
C01956=-2205,59986,1965,-1103,-34771,-352
C01957=-2177,59984,1963,-1107,-34770,-363
C01958=-2177,59984,563,-1107,-34770,-363
C01959=-2141,59982,561,-1112,-34769,-377
C01960=-2141,59982,1961,-1112,-34769,-377
C01961=-1944,59971,1947,-1138,-34763,-456
C01962=-1944,59971,547,-1138,-34763,-456
C01963=-1899,59968,544,-1144,-34761,-475
C01964=-1899,59968,1944,-1144,-34761,-475
C01965=-1684,59956,1929,-1173,-34755,-561
C01966=-1684,59956,529,-1173,-34755,-561
C01967=-1613,59952,524,-1182,-34752,-589
C01968=-1613,59952,1924,-1182,-34752,-589
C01969=-1448,59942,1913,-1204,-34747,-655
C01970=-1448,59942,513,-1204,-34747,-655
C01971=-1406,59940,510,-1209,-34746,-672
C01972=-1406,59940,1910,-1209,-34746,-672
C01973=-1043,59919,1885,-1258,-34735,-818
C01974=-1043,59919,485,-1258,-34735,-818
C01975=-1004,59917,482,-1263,-34733,-833
C01976=-1004,59917,1882,-1263,-34733,-833
C01977=-962,59914,1879,-1268,-34732,-850
C01978=-962,59914,479,-1268,-34732,-850
C01979=-945,59913,478,-1271,-34732,-857
C01980=-945,59913,1878,-1271,-34732,-857
C01981=-881,59910,1874,-1279,-34730,-883
C01982=-881,59910,474,-1279,-34730,-883
C01983=-755,59903,465,-1296,-34726,-934
C01984=-755,59903,1865,-1296,-34726,-934
C01985=-297,59876,1833,-1357,-34711,-1117
C01986=-297,59876,433,-1357,-34711,-1117
C01987=-117,59866,421,-1380,-34706,-1189
C01988=-117,59866,1821,-1380,-34706,-1189
C01989=118,59853,1805,-1412,-34699,-1284
C01990=118,59853,405,-1412,-34699,-1284
C01991=157,59850,402,-1417,-34697,-1299
C01992=157,59850,1802,-1417,-34697,-1299
C01993=231,59846,1797,-1427,-34695,-1329
C01994=231,59846,397,-1427,-34695,-1329
C01995=263,59844,395,-1431,-34694,-1342
C01996=263,59844,1795,-1431,-34694,-1342
C01997=414,59836,1784,-1451,-34689,-1402
C01998=414,59836,384,-1451,-34689,-1402
C01999=463,59833,381,-1457,-34688,-1422
C02000=463,59833,1781,-1457,-34688,-1422
C02001=597,59825,1771,-1475,-34684,-1476
C02002=597,59825,371,-1475,-34684,-1476
C02003=636,59823,369,-1480,-34682,-1491
C02004=636,59823,1769,-1480,-34682,-1491
C02005=741,59817,1761,-1494,-34679,-1533
C02006=741,59817,361,-1494,-34679,-1533
C02007=780,59815,359,-1499,-34678,-1549
C02008=780,59815,1759,-1499,-34678,-1549
C02009=1523,59772,1707,-1598,-34655,-1847
C02010=1523,59772,307,-1598,-34655,-1847
C02011=1565,59770,304,-1604,-34654,-1864
C02012=1565,59770,1704,-1604,-34654,-1864
C02013=-5497,60129,2126,-667,-34846,969
C02014=-5497,60129,726,-667,-34846,969
C02015=-5451,60127,723,-673,-34845,950
C02016=-5451,60127,2123,-673,-34845,950
C02017=-3223,59999,1969,-969,-34775,57
C02018=-3223,59999,569,-969,-34775,57
C02019=-3184,59997,566,-974,-34774,41
C02020=-3184,59997,1966,-974,-34774,41
C02021=-2783,59974,1938,-1027,-34762,-120
C02022=-2783,59974,538,-1027,-34762,-120
C02023=-2684,59969,531,-1041,-34759,-159
C02024=-2684,59969,1931,-1041,-34759,-159
C02025=-2547,59961,1922,-1059,-34754,-214
C02026=-2547,59961,522,-1059,-34754,-214
C02027=-2505,59958,519,-1064,-34753,-231
C02028=-2505,59958,1919,-1064,-34753,-231
C02029=-2244,59944,1901,-1099,-34745,-336
C02030=-2244,59944,501,-1099,-34745,-336
C02031=-2199,59941,498,-1105,-34744,-354
C02032=-2199,59941,1898,-1105,-34744,-354
C02033=-2184,59940,1897,-1107,-34743,-360
C02034=-2184,59940,497,-1107,-34743,-360
C02035=-2149,59938,494,-1112,-34742,-374
C02036=-2149,59938,1894,-1112,-34742,-374
C02037=-1952,59927,1881,-1138,-34736,-453
C02038=-1952,59927,481,-1138,-34736,-453
C02039=-1910,59924,478,-1143,-34735,-470
C02040=-1910,59924,1878,-1143,-34735,-470
C02041=-1681,59911,1862,-1174,-34727,-561
C02042=-1681,59911,462,-1174,-34727,-561
C02043=-1611,59907,457,-1183,-34725,-590
C02044=-1611,59907,1857,-1183,-34725,-590
C02045=-1452,59898,1846,-1204,-34720,-653
C02046=-1452,59898,446,-1204,-34720,-653
C02047=-1410,59896,443,-1210,-34719,-670
C02048=-1410,59896,1843,-1210,-34719,-670
C02049=-1054,59876,1819,-1257,-34708,-813
C02050=-1054,59876,419,-1257,-34708,-813
C02051=-1016,59873,416,-1262,-34707,-828
C02052=-1016,59873,1816,-1262,-34707,-828
C02053=-973,59871,1813,-1268,-34705,-845
C02054=-973,59871,413,-1268,-34705,-845
C02055=-826,59862,403,-1287,-34701,-904
C02056=-826,59862,1803,-1287,-34701,-904
C02057=-160,59824,1757,-1375,-34680,-1171
C02058=-160,59824,357,-1375,-34680,-1171
C02059=-122,59822,354,-1381,-34679,-1187
C02060=-122,59822,1754,-1381,-34679,-1187
C02061=125,59808,1737,-1413,-34671,-1286
C02062=125,59808,337,-1413,-34671,-1286
C02063=164,59806,334,-1418,-34670,-1301
C02064=164,59806,1734,-1418,-34670,-1301
C02065=216,59803,1731,-1425,-34668,-1322
C02066=216,59803,331,-1425,-34668,-1322
C02067=248,59801,329,-1430,-34667,-1335
C02068=248,59801,1729,-1430,-34667,-1335
C02069=435,59790,1716,-1454,-34662,-1410
C02070=435,59790,316,-1454,-34662,-1410
C02071=477,59788,313,-1460,-34660,-1427
C02072=477,59788,1713,-1460,-34660,-1427
C02073=604,59781,1704,-1477,-34656,-1478
C02074=604,59781,304,-1477,-34656,-1478
C02075=642,59779,301,-1482,-34655,-1493
C02076=642,59779,1701,-1482,-34655,-1493
C02077=748,59773,1694,-1496,-34652,-1535
C02078=748,59773,294,-1496,-34652,-1535
C02079=797,59770,291,-1503,-34650,-1555
C02080=797,59770,1691,-1503,-34650,-1555
C02081=1508,59729,1641,-1597,-34628,-1840
C02082=1508,59729,241,-1597,-34628,-1840
C02083=1551,59727,239,-1602,-34627,-1857
C02084=1551,59727,1639,-1602,-34627,-1857
C02085=-5487,60084,2058,-669,-34819,965
C02086=-5487,60084,658,-669,-34819,965
C02087=-5442,60082,655,-675,-34818,947
C02088=-5442,60082,2055,-675,-34818,947
C02089=-3234,59956,1902,-968,-34749,62
C02090=-3234,59956,502,-968,-34749,62
C02091=-3189,59953,499,-974,-34747,44
C02092=-3189,59953,1899,-974,-34747,44
C02093=-2544,59916,1855,-1060,-34727,-215
C02094=-2544,59916,455,-1060,-34727,-215
C02095=-2502,59914,452,-1065,-34726,-232
C02096=-2502,59914,1852,-1065,-34726,-232
C02097=-2242,59899,1834,-1100,-34718,-336
C02098=-2242,59899,434,-1100,-34718,-336
C02099=-2161,59895,428,-1111,-34715,-369
C02100=-2161,59895,1828,-1111,-34715,-369
C02101=-1963,59883,1815,-1137,-34709,-448
C02102=-1963,59883,415,-1137,-34709,-448
C02103=-1918,59881,411,-1143,-34708,-466
C02104=-1918,59881,1811,-1143,-34708,-466
C02105=-1678,59867,1795,-1175,-34700,-562
C02106=-1678,59867,395,-1175,-34700,-562
C02107=-1601,59863,390,-1185,-34698,-593
C02108=-1601,59863,1790,-1185,-34698,-593
C02109=-1457,59854,1780,-1204,-34693,-651
C02110=-1457,59854,380,-1204,-34693,-651
C02111=-1414,59852,377,-1210,-34692,-668
C02112=-1414,59852,1777,-1210,-34692,-668
C02113=-1062,59832,1752,-1257,-34681,-809
C02114=-1062,59832,352,-1257,-34681,-809
C02115=-1024,59830,350,-1262,-34680,-824
C02116=-1024,59830,1750,-1262,-34680,-824
C02117=-154,59780,1689,-1377,-34653,-1173
C02118=-154,59780,289,-1377,-34653,-1173
C02119=-115,59778,287,-1382,-34652,-1189
C02120=-115,59778,1687,-1382,-34652,-1189
C02121=131,59764,1670,-1415,-34644,-1288
C02122=131,59764,270,-1415,-34644,-1288
C02123=173,59761,267,-1421,-34643,-1304
C02124=173,59761,1667,-1421,-34643,-1304
C02125=205,59760,1665,-1425,-34642,-1317
C02126=205,59760,265,-1425,-34642,-1317
C02127=237,59758,262,-1429,-34641,-1330
C02128=237,59758,1662,-1429,-34641,-1330
C02129=448,59746,1648,-1457,-34634,-1415
C02130=448,59746,248,-1457,-34634,-1415
C02131=490,59743,245,-1463,-34633,-1431
C02132=490,59743,1645,-1463,-34633,-1431
C02133=606,59737,1637,-1478,-34629,-1478
C02134=606,59737,237,-1478,-34629,-1478
C02135=649,59734,234,-1484,-34628,-1495
C02136=649,59734,1634,-1484,-34628,-1495
C02137=765,59728,1626,-1499,-34624,-1542
C02138=765,59728,226,-1499,-34624,-1542
C02139=856,59722,220,-1511,-34621,-1578
C02140=856,59722,1620,-1511,-34621,-1578
C02141=1494,59686,1575,-1596,-34601,-1834
C02142=1494,59686,175,-1596,-34601,-1834
C02143=1536,59684,173,-1601,-34600,-1851
C02144=1536,59684,1573,-1601,-34600,-1851
C02145=-5481,60040,1991,-671,-34792,964
C02146=-5481,60040,591,-671,-34792,964
C02147=-5429,60037,587,-678,-34790,942
C02148=-5429,60037,1987,-678,-34790,942
C02149=-3242,59912,1836,-968,-34722,66
C02150=-3242,59912,436,-968,-34722,66
C02151=-3200,59910,433,-973,-34721,49
C02152=-3200,59910,1833,-973,-34721,49
C02153=-2545,59872,1788,-1060,-34700,-214
C02154=-2545,59872,388,-1060,-34700,-214
C02155=-2503,59870,385,-1066,-34699,-231
C02156=-2503,59870,1785,-1066,-34699,-231
C02157=-2235,59855,1766,-1102,-34691,-338
C02158=-2235,59855,366,-1102,-34691,-338
C02159=-2165,59851,361,-1111,-34688,-366
C02160=-2165,59851,1761,-1111,-34688,-366
C02161=-1964,59839,1748,-1138,-34682,-447
C02162=-1964,59839,348,-1138,-34682,-447
C02163=-1926,59837,345,-1143,-34681,-462
C02164=-1926,59837,1745,-1143,-34681,-462
C02165=-1679,59823,1728,-1175,-34673,-561
C02166=-1679,59823,328,-1175,-34673,-561
C02167=-1595,59818,322,-1187,-34671,-595
C02168=-1595,59818,1722,-1187,-34671,-595
C02169=-1457,59810,1713,-1205,-34666,-650
C02170=-1457,59810,313,-1205,-34666,-650
C02171=-1415,59808,310,-1210,-34665,-667
C02172=-1415,59808,1710,-1210,-34665,-667
C02173=-1070,59788,1686,-1256,-34654,-805
C02174=-1070,59788,286,-1256,-34654,-805
C02175=-1028,59786,283,-1262,-34653,-822
C02176=-1028,59786,1683,-1262,-34653,-822
C02177=-148,59736,1622,-1379,-34625,-1175
C02178=-148,59736,222,-1379,-34625,-1175
C02179=-109,59733,219,-1384,-34624,-1191
C02180=-109,59733,1619,-1384,-34624,-1191
C02181=141,59719,1602,-1417,-34616,-1291
C02182=141,59719,202,-1417,-34616,-1291
C02183=180,59717,199,-1422,-34615,-1306
C02184=180,59717,1599,-1422,-34615,-1306
C02185=194,59716,1598,-1424,-34615,-1312
C02186=194,59716,198,-1424,-34615,-1312
C02187=226,59714,196,-1428,-34614,-1325
C02188=226,59714,1596,-1428,-34614,-1325
C02189=461,59701,1580,-1460,-34606,-1419
C02190=461,59701,180,-1460,-34606,-1419
C02191=500,59699,177,-1465,-34605,-1435
C02192=500,59699,1577,-1465,-34605,-1435
C02193=613,59692,1569,-1480,-34602,-1480
C02194=613,59692,169,-1480,-34602,-1480
C02195=659,59690,166,-1486,-34600,-1498
C02196=659,59690,1566,-1486,-34600,-1498
C02197=803,59681,1556,-1505,-34596,-1556
C02198=803,59681,156,-1505,-34596,-1556
C02199=1071,59666,138,-1540,-34587,-1664
C02200=1071,59666,1538,-1540,-34587,-1664
C02201=1479,59643,1509,-1595,-34575,-1827
C02202=1479,59643,109,-1595,-34575,-1827
C02203=1525,59640,106,-1601,-34573,-1846
C02204=1525,59640,1506,-1601,-34573,-1846
C02205=-5472,59994,1923,-673,-34765,960
C02206=-5472,59994,523,-673,-34765,960
C02207=-5419,59991,519,-680,-34763,939
C02208=-5419,59991,1919,-680,-34763,939
C02209=-3254,59868,1770,-967,-34695,71
C02210=-3254,59868,370,-967,-34695,71
C02211=-3208,59866,367,-973,-34694,53
C02212=-3208,59866,1767,-973,-34694,53
C02213=-2542,59828,1721,-1061,-34673,-214
C02214=-2542,59828,321,-1061,-34673,-214
C02215=-2500,59825,318,-1067,-34672,-231
C02216=-2500,59825,1718,-1067,-34672,-231
C02217=-2229,59810,1699,-1103,-34663,-340
C02218=-2229,59810,299,-1103,-34663,-340
C02219=-2166,59806,295,-1112,-34661,-365
C02220=-2166,59806,1695,-1112,-34661,-365
C02221=-1972,59795,1681,-1137,-34655,-443
C02222=-1972,59795,281,-1137,-34655,-443
C02223=-1926,59793,278,-1143,-34654,-461
C02224=-1926,59793,1678,-1143,-34654,-461
C02225=-1683,59779,1661,-1176,-34646,-559
C02226=-1683,59779,261,-1176,-34646,-559
C02227=-1655,59777,259,-1179,-34645,-570
C02228=-1655,59777,1659,-1179,-34645,-570
C02229=-1634,59776,1658,-1182,-34645,-578
C02230=-1634,59776,258,-1182,-34645,-578
C02231=-1592,59774,255,-1188,-34643,-595
C02232=-1592,59774,1655,-1188,-34643,-595
C02233=-1455,59766,1645,-1206,-34639,-650
C02234=-1455,59766,245,-1206,-34639,-650
C02235=-1419,59764,243,-1211,-34638,-665
C02236=-1419,59764,1643,-1211,-34638,-665
C02237=-1067,59744,1619,-1257,-34627,-806
C02238=-1067,59744,219,-1257,-34627,-806
C02239=-1032,59742,216,-1262,-34626,-820
C02240=-1032,59742,1616,-1262,-34626,-820
C02241=-145,59691,1555,-1380,-34598,-1176
C02242=-145,59691,155,-1380,-34598,-1176
C02243=-106,59689,152,-1385,-34597,-1191
C02244=-106,59689,1552,-1385,-34597,-1191
C02245=147,59675,1535,-1419,-34589,-1293
C02246=147,59675,135,-1419,-34589,-1293
C02247=221,59671,129,-1428,-34587,-1322
C02248=221,59671,1529,-1428,-34587,-1322
C02249=471,59656,1512,-1462,-34579,-1423
C02250=471,59656,112,-1462,-34579,-1423
C02251=510,59654,109,-1467,-34578,-1438
C02252=510,59654,1509,-1467,-34578,-1438
C02253=623,59648,1502,-1482,-34574,-1483
C02254=623,59648,102,-1482,-34574,-1483
C02255=665,59645,99,-1487,-34573,-1500
C02256=665,59645,1499,-1487,-34573,-1500
C02257=1010,59626,1475,-1533,-34562,-1639
C02258=1010,59626,75,-1533,-34562,-1639
C02259=1137,59618,66,-1550,-34558,-1689
C02260=1137,59618,1466,-1550,-34558,-1689
C02261=1468,59600,1443,-1594,-34548,-1822
C02262=1468,59600,43,-1594,-34548,-1822
C02263=1517,59597,40,-1600,-34546,-1842
C02264=1517,59597,1440,-1600,-34546,-1842
C02265=-5459,59949,1855,-675,-34737,955
C02266=-5459,59949,455,-675,-34737,955
C02267=-5409,59946,452,-682,-34736,936
C02268=-5409,59946,1852,-682,-34736,936
C02269=-3269,59825,1704,-966,-34669,77
C02270=-3269,59825,304,-966,-34669,77
C02271=-3216,59822,300,-973,-34667,56
C02272=-3216,59822,1700,-973,-34667,56
C02273=-2540,59783,1653,-1063,-34646,-215
C02274=-2540,59783,253,-1063,-34646,-215
C02275=-2501,59781,251,-1068,-34645,-230
C02276=-2501,59781,1651,-1068,-34645,-230
C02277=-2230,59766,1632,-1104,-34636,-339
C02278=-2230,59766,232,-1104,-34636,-339
C02279=-2170,59762,228,-1112,-34634,-363
C02280=-2170,59762,1628,-1112,-34634,-363
C02281=-1966,59751,1614,-1139,-34628,-445
C02282=-1966,59751,214,-1139,-34628,-445
C02283=-1924,59748,211,-1144,-34627,-462
C02284=-1924,59748,1611,-1144,-34627,-462
C02285=-1688,59735,1594,-1176,-34619,-556
C02286=-1688,59735,194,-1176,-34619,-556
C02287=-1656,59733,192,-1180,-34618,-569
C02288=-1656,59733,1592,-1180,-34618,-569
C02289=-1628,59732,1590,-1184,-34617,-580
C02290=-1628,59732,190,-1184,-34617,-580
C02291=-1582,59729,187,-1190,-34616,-599
C02292=-1582,59729,1587,-1190,-34616,-599
C02293=-1452,59722,1578,-1207,-34612,-651
C02294=-1452,59722,178,-1207,-34612,-651
C02295=-1410,59719,175,-1213,-34611,-668
C02296=-1410,59719,1575,-1213,-34611,-668
C02297=-1068,59700,1552,-1258,-34600,-805
C02298=-1068,59700,152,-1258,-34600,-805
C02299=-1033,59698,149,-1263,-34599,-819
C02300=-1033,59698,1549,-1263,-34599,-819
C02301=-138,59647,1487,-1381,-34571,-1178
C02302=-138,59647,87,-1381,-34571,-1178
C02303=-100,59645,85,-1387,-34570,-1193
C02304=-100,59645,1485,-1387,-34570,-1193
C02305=157,59630,1467,-1421,-34562,-1296
C02306=157,59630,67,-1421,-34562,-1296
C02307=217,59627,63,-1429,-34560,-1320
C02308=217,59627,1463,-1429,-34560,-1320
C02309=478,59612,1445,-1463,-34551,-1425
C02310=478,59612,45,-1463,-34551,-1425
C02311=520,59610,42,-1469,-34550,-1442
C02312=520,59610,1442,-1469,-34550,-1442
C02313=629,59603,1434,-1483,-34547,-1485
C02314=629,59603,34,-1483,-34547,-1485
C02315=671,59601,31,-1489,-34545,-1502
C02316=671,59601,1431,-1489,-34545,-1502
C02317=1112,59576,1401,-1547,-34532,-1679
C02318=1112,59576,1,-1547,-34532,-1679
C02319=1178,59572,-4,-1556,-34530,-1706
C02320=1178,59572,1396,-1556,-34530,-1706
C02321=1457,59556,1377,-1593,-34521,-1817
C02322=1457,59556,-23,-1593,-34521,-1817
C02323=1499,59554,-26,-1599,-34520,-1834
C02324=1499,59554,1374,-1599,-34520,-1834
C02325=-5446,59904,1787,-677,-34710,951
C02326=-5446,59904,387,-677,-34710,951
C02327=-5396,59901,384,-684,-34708,931
C02328=-5396,59901,1784,-684,-34708,931
C02329=-4572,59854,1727,-793,-34683,601
C02330=-4572,59854,327,-793,-34683,601
C02331=-4520,59851,323,-800,-34681,579
C02332=-4520,59851,1723,-800,-34681,579
C02333=-4111,59828,1695,-855,-34668,416
C02334=-4111,59828,295,-855,-34668,416
C02335=-4094,59827,294,-857,-34668,409
C02336=-4094,59827,1694,-857,-34668,409
C02337=-3284,59781,1638,-965,-34642,84
C02338=-3284,59781,238,-965,-34642,84
C02339=-3234,59779,234,-971,-34641,64
C02340=-3234,59779,1634,-971,-34641,64
C02341=-2541,59739,1586,-1063,-34619,-214
C02342=-2541,59739,186,-1063,-34619,-214
C02343=-2502,59737,184,-1068,-34618,-229
C02344=-2502,59737,1584,-1068,-34618,-229
C02345=-2227,59721,1565,-1105,-34609,-340
C02346=-2227,59721,165,-1105,-34609,-340
C02347=-2174,59718,161,-1112,-34607,-361
C02348=-2174,59718,1561,-1112,-34607,-361
C02349=-1963,59706,1546,-1140,-34601,-445
C02350=-1963,59706,146,-1140,-34601,-445
C02351=-1921,59704,144,-1145,-34600,-462
C02352=-1921,59704,1544,-1145,-34600,-462
C02353=-1696,59691,1528,-1175,-34592,-553
C02354=-1696,59691,128,-1175,-34592,-553
C02355=-1664,59689,126,-1180,-34591,-565
C02356=-1664,59689,1526,-1180,-34591,-565
C02357=-1622,59687,1523,-1185,-34590,-582
C02358=-1622,59687,123,-1185,-34590,-582
C02359=-1576,59684,120,-1191,-34589,-601
C02360=-1576,59684,1520,-1191,-34589,-601
C02361=-1446,59677,1511,-1209,-34585,-653
C02362=-1446,59677,111,-1209,-34585,-653
C02363=-1400,59674,107,-1215,-34583,-671
C02364=-1400,59674,1507,-1215,-34583,-671
C02365=-1065,59656,1484,-1259,-34573,-805
C02366=-1065,59656,84,-1259,-34573,-805
C02367=-1030,59654,82,-1264,-34572,-819
C02368=-1030,59654,1482,-1264,-34572,-819
C02369=-136,59603,1420,-1383,-34544,-1178
C02370=-136,59603,20,-1383,-34544,-1178
C02371=-100,59601,18,-1387,-34542,-1192
C02372=-100,59601,1418,-1387,-34542,-1192
C02373=164,59586,1399,-1422,-34534,-1298
C02374=164,59586,-1,-1422,-34534,-1298
C02375=217,59583,-4,-1429,-34533,-1319
C02376=217,59583,1396,-1429,-34533,-1319
C02377=484,59568,1377,-1465,-34524,-1427
C02378=484,59568,-23,-1465,-34524,-1427
C02379=526,59565,-26,-1470,-34523,-1443
C02380=526,59565,1374,-1470,-34523,-1443
C02381=632,59559,1367,-1485,-34519,-1486
C02382=632,59559,-33,-1485,-34519,-1486
C02383=674,59557,-36,-1490,-34518,-1503
C02384=674,59557,1364,-1490,-34518,-1503
C02385=1150,59530,1331,-1553,-34503,-1693
C02386=1150,59530,-69,-1553,-34503,-1693
C02387=1199,59527,-72,-1560,-34502,-1713
C02388=1199,59527,1328,-1560,-34502,-1713
C02389=-5436,59859,1719,-679,-34683,947
C02390=-5436,59859,319,-679,-34683,947
C02391=-5383,59856,316,-686,-34681,926
C02392=-5383,59856,1716,-686,-34681,926
C02393=-4577,59810,1660,-793,-34656,603
C02394=-4577,59810,260,-793,-34656,603
C02395=-4521,59807,256,-801,-34654,580
C02396=-4521,59807,1656,-801,-34654,580
C02397=-4144,59786,1630,-851,-34642,429
C02398=-4144,59786,230,-851,-34642,429
C02399=-4087,59783,226,-858,-34640,407
C02400=-4087,59783,1626,-858,-34640,407
C02401=-3299,59738,1572,-963,-34616,91
C02402=-3299,59738,172,-963,-34616,91
C02403=-3253,59735,168,-969,-34614,72
C02404=-3253,59735,1568,-969,-34614,72
C02405=-2541,59695,1519,-1064,-34592,-213
C02406=-2541,59695,119,-1064,-34592,-213
C02407=-2503,59693,117,-1069,-34591,-228
C02408=-2503,59693,1517,-1069,-34591,-228
C02409=-2225,59677,1497,-1106,-34582,-340
C02410=-2225,59677,97,-1106,-34582,-340
C02411=-2175,59674,94,-1112,-34580,-360
C02412=-2175,59674,1494,-1112,-34580,-360
C02413=-1953,59662,1479,-1142,-34573,-449
C02414=-1953,59662,79,-1142,-34573,-449
C02415=-1908,59659,76,-1148,-34572,-467
C02416=-1908,59659,1476,-1148,-34572,-467
C02417=-1707,59648,1462,-1175,-34566,-548
C02418=-1707,59648,62,-1175,-34566,-548
C02419=-1675,59646,59,-1179,-34565,-560
C02420=-1675,59646,1459,-1179,-34565,-560
C02421=-1612,59642,1455,-1187,-34563,-586
C02422=-1612,59642,55,-1187,-34563,-586
C02423=-1570,59640,52,-1193,-34561,-603
C02424=-1570,59640,1452,-1193,-34561,-603
C02425=-1429,59632,1442,-1212,-34557,-659
C02426=-1429,59632,42,-1212,-34557,-659
C02427=-1386,59630,40,-1217,-34556,-676
C02428=-1386,59630,1440,-1217,-34556,-676
C02429=-1168,59617,1424,-1246,-34549,-764
C02430=-1168,59617,24,-1246,-34549,-764
C02431=-1122,59615,21,-1252,-34547,-782
C02432=-1122,59615,1421,-1252,-34547,-782
C02433=-1062,59611,1417,-1260,-34545,-806
C02434=-1062,59611,17,-1260,-34545,-806
C02435=-1024,59609,14,-1265,-34544,-821
C02436=-1024,59609,1414,-1265,-34544,-821
C02437=-629,59587,1387,-1318,-34532,-980
C02438=-629,59587,-13,-1318,-34532,-980
